// TIA Portal V20 export
FUNCTION_BLOCK "CallEquipment"   // FB32, LAD
TITLE = CallEquipment
AUTHOR : ERsystem_FA2_DH. Kim
// This block contains the logic and futher calls (e.g. sequences, control modules, diagnostics etc.) of the equipment module.
// stored: IsIECCheckEnabled true, MemoryReserve 100, Namespace Unit1.Em4, SetENOAutomatically false
   VAR_INPUT
      ZoneOperationEnable { ExternalWritable := 'False'} : "LWONIK_typeSafetyZoneManualOperation";
   END_VAR
   VAR_IN_OUT
      unitStatus : "LAF_typeUnitStatus";   // Current unit status o be used in this EM
      unitAlarmDB : "LAF_typeAlarms";   // Summarized EM Alarms for the Unit
      emFeedback : "LUC_typeEmFeedback";   // Feedback of the EM to the Unit
   END_VAR
   VAR
      InstSequenceMainPnP : "Unit1.Em4.Sequence_1_MainPnP";   // EM Sequence Instance
      InstSequenceAlignTable : "Unit1.Em4.Sequence_2_AlignTable";
      InstSequenceNgPnP : "Unit1.Em4.Sequence_3_NgPnP";
      InstSequenceGaugeRnR : "Unit1.Em4.Sequence_10_GaugeRnR";
      instMainPnPHomeJob1 : "LAF_SelectJob";
      instMainPnPHomeJob10 : "LAF_SelectJob";
      instMainPnPLoadJob2 : "LAF_SelectJob";
      instMainPnPUnloadJob3 : "LAF_SelectJob";
      instMainPnPAvoidJob4 : "LAF_SelectJob";
      instMainPnPOneLoadJob5 : "LAF_SelectJob";
      instMainPnPOneUnLoadJob6 : "LAF_SelectJob";
      instMainPnPDownWaitJob7 { S7_SetPoint := 'True'} : "LAF_SelectJob";
      instAlignTableHomeJob1 : "LAF_SelectJob";
      instAlignTableLoadJob2 : "LAF_SelectJob";
      instAlignTableVisionJob3 : "LAF_SelectJob";
      instAlignTableUnloadJob4 : "LAF_SelectJob";
      instAlignTableMotionJob22 : "LAF_SelectJob";
      instNgPnPHomeJob1 : "LAF_SelectJob";
      instNgPnPLoadJob2 : "LAF_SelectJob";
      instNgPnPUnloadJob3 : "LAF_SelectJob";
      instGaugeRnRCommonReadyJob1 : "LAF_SelectJob";
      instGaugeRnRCommonGetMasterPieceJob2 : "LAF_SelectJob";
      instGaugeRnRCommonMainPnPMoveAlignTableStackTableJob3 : "LAF_SelectJob";
      instGaugeRnRCommonMainPnp1ToAlignTableJob4 : "LAF_SelectJob";
      instGaugeRnRCommonMainPnPMoveReelCutConvyorAlignTableJob5 : "LAF_SelectJob";
      instGaugeRnRCommonAlignTableVisionAdjustJob6 : "LAF_SelectJob";
      instGaugeRnR1AlignAlignTableToMainPnP1Job10 { S7_SetPoint := 'True'} : "LAF_SelectJob";
      instGaugeRnR1AlignMainPnPMoveReelCutConvyorAlignTableJob11 { S7_SetPoint := 'True'} : "LAF_SelectJob";
      instGaugeRnR1AlignAlignTableMoveWaitJob12 { S7_SetPoint := 'True'} : "LAF_SelectJob";
      instGaugeRnR1AlignUnloadMasterPieceJob13 { S7_SetPoint := 'True'} : "LAF_SelectJob";
      instGaugeRnR1StackMainPnPMoveReelCutConvyorAlignTableJob15 { S7_SetPoint := 'True'} : "LAF_SelectJob";
      instGaugeRnR1StackAlignTableToMainPnP2Job16 { S7_SetPoint := 'True'} : "LAF_SelectJob";
      instGaugeRnR1StackMainPnPMoveAlignTableJob17 { S7_SetPoint := 'True'} : "LAF_SelectJob";
      instGaugeRnR1StackAlignTableMoveWaitJob18 { S7_SetPoint := 'True'} : "LAF_SelectJob";
      instGaugeRnR1StackMainPnP2ToStackTableJob19 { S7_SetPoint := 'True'} : "LAF_SelectJob";
      instGaugeRnR1StackStackTableToMainPnP2Job20 { S7_SetPoint := 'True'} : "LAF_SelectJob";
      instGaugeRnR1StackMainPnPMoveReelCutConvyorAlignTableJob21 { S7_SetPoint := 'True'} : "LAF_SelectJob";
      instGaugeRnR1StackMainPnP2ToAlignTableJob22 { S7_SetPoint := 'True'} : "LAF_SelectJob";
      instGaugeRnR1StackMainPnPMoveAlignTableJob23 { S7_SetPoint := 'True'} : "LAF_SelectJob";
      instGaugeRnR1StackAlignTableToMainPnP1Job24 { S7_SetPoint := 'True'} : "LAF_SelectJob";
      instGaugeRnR1StackMainPnPMoveReelCutConvyorAlignTableJob25 { S7_SetPoint := 'True'} : "LAF_SelectJob";
      instGaugeRnR1StackUnloadMasterPieceJob26 { S7_SetPoint := 'True'} : "LAF_SelectJob";
      instGaugeRnR3AlignMainPnPMoveReelCutConvyorAlignTableJob30 { S7_SetPoint := 'True'} : "LAF_SelectJob";
      instGaugeRnR3AlignNGPnPLoadMasterPieceJob31 { S7_SetPoint := 'True'} : "LAF_SelectJob";
      instGaugeRnR3AlignMainPnP2MoveAlignTableJob32 { S7_SetPoint := 'True'} : "LAF_SelectJob";
      instGaugeRnR3AlignAlignTableMoveWaitJob33 { S7_SetPoint := 'True'} : "LAF_SelectJob";
      instGaugeRnRCommonCheckCompleteJob39 { S7_SetPoint := 'True'} : "LAF_SelectJob";
      instCmPnp1stAnodeDetectSensor { S7_SetPoint := 'True'} : "LBC_DigitalSignalCn";
      instCmPnp2ndAnodeDetectSensor { S7_SetPoint := 'True'} : "LBC_DigitalSignalCn";
      instCmAnodeAlignTableElectrodeDetectSensor { S7_SetPoint := 'True'} : "LBC_DigitalSignalCn";
      instCmAnodeNgBoxFullSensorDetectSensor { S7_SetPoint := 'True'} : "LBC_DigitalSignalCn";
      instCmAnodeNgBoxDetectSensor { S7_SetPoint := 'True'} : "LBC_DigitalSignalCn";
      instCmAnodeMainPnP1AxisX { S7_SetPoint := 'True'} : "LBC_Axis64Pos_TecPlcCn";   // Axis 64Position Function Block
      instCmAnodeMainPnP2AxisX { S7_SetPoint := 'True'} : "LBC_Axis64Pos_TecPlcCn";   // Axis 64Position Function Block
      instCmAnodeMainPnP1AxisY { S7_SetPoint := 'True'} : "LBC_Axis64Pos_TecPlcCn";   // Axis 64Position Function Block
      instCmAnodeMainPnP1AxisZ { S7_SetPoint := 'True'} : "LBC_Axis64Pos_TecPlcCn";   // Axis 64Position Function Block
      instCmAnodeMainPnP2AxisZ { S7_SetPoint := 'True'} : "LBC_Axis64Pos_TecPlcCn";   // Axis 64Position Function Block
      instCmAnodeAlignTableAxisX { S7_SetPoint := 'True'} : "LBC_Axis64Pos_TecPlcCn";   // Axis 64Position Function Block
      instCmAnodeAlignTableAxisY1 { S7_SetPoint := 'True'} : "LBC_Axis64Pos_TecPlcCn";   // Axis 64Position Function Block
      instCmAnodeAlignTableAxisY2 { S7_SetPoint := 'True'} : "LBC_Axis64Pos_TecPlcCn";   // Axis 64Position Function Block
      instInterlockAnodeMainPnP1AxisX { S7_SetPoint := 'True'} : "LER_Axis64Pos_InterlockSummary";
      instInterlockAnodeMainPnP1AxisY { S7_SetPoint := 'True'} : "LER_Axis64Pos_InterlockSummary";
      instInterlockAnodeMainPnP1AxisZ { S7_SetPoint := 'True'} : "LER_Axis64Pos_InterlockSummary";
      instInterlockAnodeMainPnP2AxisX { S7_SetPoint := 'True'} : "LER_Axis64Pos_InterlockSummary";
      instInterlockAnodeMainPnP2AxisZ { S7_SetPoint := 'True'} : "LER_Axis64Pos_InterlockSummary";
      instInterlockAnodeAlignTableAxisX { S7_SetPoint := 'True'} : "LER_Axis64Pos_InterlockSummary";
      instInterlockAnodeAlignTableAxisY1 { S7_SetPoint := 'True'} : "LER_Axis64Pos_InterlockSummary";
      instInterlockAnodeAlignTableAxisY2 { S7_SetPoint := 'True'} : "LER_Axis64Pos_InterlockSummary";
      instAnodeMainPnP1AxisXSoftCam : "LER_SoftCam_Interface";
      instAnodeMainPnP2AxisXSoftCam { S7_SetPoint := 'True'} : "LER_SoftCam_Interface";
      instAnodeMainPnP1AxisYSoftCam { S7_SetPoint := 'True'} : "LER_SoftCam_Interface";
      instAnodeMainPnP1AxisZSoftCam { S7_SetPoint := 'True'} : "LER_SoftCam_Interface";
      instAnodeMainPnP2AxisZSoftCam { S7_SetPoint := 'True'} : "LER_SoftCam_Interface";
      instAnodeAlignTableAxisXSoftCam { S7_SetPoint := 'True'} : "LER_SoftCam_Interface";
      instAnodeAlignTableAxisY1SoftCam { S7_SetPoint := 'True'} : "LER_SoftCam_Interface";
      instAnodeAlignTableAxisY2SoftCam { S7_SetPoint := 'True'} : "LER_SoftCam_Interface";
      instCmAnodeMainPnP1RotaryCwCcw { ExternalAccessible := 'False'; ExternalVisible := 'False'; ExternalWritable := 'False'} : "LBC_TwoWayActuatorCn";
      instCmAnodeMainPnP1stSuctionPlateVacuum { ExternalAccessible := 'False'; ExternalVisible := 'False'; ExternalWritable := 'False'} : "LBC_TwoWayActuatorCn";
      instCmAnodeMainPnP2ndSuctionPlateVacuum { ExternalAccessible := 'False'; ExternalVisible := 'False'; ExternalWritable := 'False'} : "LBC_TwoWayActuatorCn";
      instCmAnodeAlignTableSuctionPlateVacuum { ExternalAccessible := 'False'; ExternalVisible := 'False'; ExternalWritable := 'False'; S7_SetPoint := 'True'} : "LBC_TwoWayActuatorCn";
      instCmAnodeGlassCleaning { ExternalAccessible := 'False'; ExternalVisible := 'False'; ExternalWritable := 'False'; S7_SetPoint := 'True'} : "LBC_TwoWayActuatorCn";
      instCmAnodeNgPnpUpDown { ExternalAccessible := 'False'; ExternalVisible := 'False'; ExternalWritable := 'False'; S7_SetPoint := 'True'} : "LBC_TwoWayActuatorCn";
      instCmAnodeNgPnp1stFwdBwd { ExternalAccessible := 'False'; ExternalVisible := 'False'; ExternalWritable := 'False'; S7_SetPoint := 'True'} : "LBC_TwoWayActuatorCn";
      instCmAnodeNgPnp2ndFwdBwd { ExternalAccessible := 'False'; ExternalVisible := 'False'; ExternalWritable := 'False'; S7_SetPoint := 'True'} : "LBC_TwoWayActuatorCn";
      instCmAnodeMaintenanceMovingFixFwdBwd { ExternalAccessible := 'False'; ExternalVisible := 'False'; ExternalWritable := 'False'; S7_SetPoint := 'True'} : "LBC_TwoWayActuatorCn";
      instCmAnodeNgBoxLiftUpDown { ExternalAccessible := 'False'; ExternalVisible := 'False'; ExternalWritable := 'False'; S7_SetPoint := 'True'} : "LBC_TwoWayActuatorCn";
      instCmAnodeNgBoxLockUpDown { ExternalAccessible := 'False'; ExternalVisible := 'False'; ExternalWritable := 'False'; S7_SetPoint := 'True'} : "LBC_TwoWayActuatorCn";
      instCmAnodeNgPnpVaccum { ExternalAccessible := 'False'; ExternalVisible := 'False'; ExternalWritable := 'False'; S7_SetPoint := 'True'} : "LBC_TwoWayActuatorCn";
      instCmAnodeConveyorCoverFwdBwd { S7_SetPoint := 'True'} : "LBC_TwoWayActuatorCn";
      instCmAnodeConveyorPickUpBlower { S7_SetPoint := 'True'} : "LBC_TwoWayActuatorCn";
      instCmAnodeVisionControllerInterface { ExternalAccessible := 'False'; ExternalVisible := 'False'; ExternalWritable := 'False'; S7_SetPoint := 'True'} : "LER_Vision_XGX2000";
      instAlignVisionConversion : "LER_AlignVisionConversion";
      instManageAlarms { ExternalWritable := 'False'} : "LAF_ManageAlarms";
      instLER_BrakeTestAnodeMainPnP1AxisZ : "LER_BrakeTest";
      instLER_BrakeTestAnodeMainPnP2AxisZ { S7_SetPoint := 'True'} : "LER_BrakeTest";
      instEventsPFE : "Unit1.Em4.EventsPFE";
      statUnitStatus { ExternalWritable := 'False'} : "LAF_typeUnitStatus";   // Unit Status used in this EM
      statSlmStatus { ExternalWritable := 'False'} : Struct
         running : Bool;
         powerOff : Bool;
      END_STRUCT;
      statAllBrakeTest { ExternalWritable := 'False'} : "LER_typeBrakeTestUnitCommands";
      statInterlockTonTime { ExternalAccessible := 'False'; ExternalVisible := 'False'; ExternalWritable := 'False'} : Struct
         mainPnP1AxisX : Array[0..15] of TON_TIME;
         mainPnP1AxisY : Array[0..15] of TON_TIME;
         mainPnP1AxisZ : Array[0..15] of TON_TIME;
         mainPnP2AxisX : Array[0..15] of TON_TIME;
         mainPnP2AxisZ : Array[0..15] of TON_TIME;
         alignTableAxisX : Array[0..15] of TON_TIME;
         alignTableAxisY1 : Array[0..15] of TON_TIME;
         alignTableAxisY2 : Array[0..15] of TON_TIME;
      END_STRUCT;
      statTonTime { ExternalAccessible := 'False'; ExternalVisible := 'False'; ExternalWritable := 'False'} : Array[0..1999] of TON_TIME;
      statTofTime { ExternalAccessible := 'False'; ExternalVisible := 'False'; ExternalWritable := 'False'} : Array[0..99] of TOF_TIME;
      statPulse { ExternalAccessible := 'False'; ExternalVisible := 'False'; ExternalWritable := 'False'} : Struct
         miscellaneous : Array[0..99] of Bool;
         workingDone : Struct
            mainPnP : Array[0..99] of Bool;
            alignTable : Array[0..99] of Bool;
            ngPnP : Array[0..99] of Bool;
         END_STRUCT;
         axisEnable : Array[0..99] of Bool;
         brakeTest : Array[0..99] of Bool;
      END_STRUCT;
      statEnableManualCmds : Bool;
      Scan_on : Bool;
      "*** Interlock Axis ***" { ExternalAccessible := 'False'; ExternalVisible := 'False'; ExternalWritable := 'False'} : Bool;
      "AnodeMainPnP1AxisX Home" { S7_SetPoint := 'True'} : "Homing.LER_Axis";
      "AnodeMainPnP1AxisX Jog_CW" { S7_SetPoint := 'True'} : "Jog.LER_Axis";
      "AnodeMainPnP1AxisX Jog_CCW" { S7_SetPoint := 'True'} : "Jog.LER_Axis";
      "AnodeMainPnP1AxisX Position_" { S7_SetPoint := 'True'} : Array[0..5] of "Position.LER_Axis";
      "AnodeMainPnP2AxisX Home" { S7_SetPoint := 'True'} : "Homing.LER_Axis";
      "AnodeMainPnP2AxisX Jog_CW" { S7_SetPoint := 'True'} : "Jog.LER_Axis";
      "AnodeMainPnP2AxisX Jog_CCW" { S7_SetPoint := 'True'} : "Jog.LER_Axis";
      "AnodeMainPnP2AxisX Position_" { S7_SetPoint := 'True'} : Array[0..5] of "Position.LER_Axis";
      "AnodeMainPnP1AxisY Home" { S7_SetPoint := 'True'} : "Homing.LER_Axis";
      "AnodeMainPnP1AxisY Jog_CW" { S7_SetPoint := 'True'} : "Jog.LER_Axis";
      "AnodeMainPnP1AxisY Jog_CCW" { S7_SetPoint := 'True'} : "Jog.LER_Axis";
      "AnodeMainPnP1AxisY Position_" { S7_SetPoint := 'True'} : Array[0..5] of "Position.LER_Axis";
      "AnodeMainPnP1AxisZ Home" { S7_SetPoint := 'True'} : "Homing.LER_Axis";
      "AnodeMainPnP1AxisZ Jog_CW" { S7_SetPoint := 'True'} : "Jog.LER_Axis";
      "AnodeMainPnP1AxisZ Jog_CCW" { S7_SetPoint := 'True'} : "Jog.LER_Axis";
      "AnodeMainPnP1AxisZ Position_" { S7_SetPoint := 'True'} : Array[0..5] of "Position.LER_Axis";
      "AnodeMainPnP2AxisZ Home" { S7_SetPoint := 'True'} : "Homing.LER_Axis";
      "AnodeMainPnP2AxisZ Jog_CW" { S7_SetPoint := 'True'} : "Jog.LER_Axis";
      "AnodeMainPnP2AxisZ Jog_CCW" { S7_SetPoint := 'True'} : "Jog.LER_Axis";
      "AnodeMainPnP2AxisZ Position_" { S7_SetPoint := 'True'} : Array[0..5] of "Position.LER_Axis";
      "AnodeAlignTableAxisX Home" { S7_SetPoint := 'True'} : "Homing.LER_Axis";
      "AnodeAlignTableAxisX Jog_CW" { S7_SetPoint := 'True'} : "Jog.LER_Axis";
      "AnodeAlignTableAxisX Jog_CCW" { S7_SetPoint := 'True'} : "Jog.LER_Axis";
      "AnodeAlignTableAxisX Position_" { S7_SetPoint := 'True'} : Array[0..5] of "Position.LER_Axis";
      "AnodeAlignTableAxisY1 Home" { S7_SetPoint := 'True'} : "Homing.LER_Axis";
      "AnodeAlignTableAxisY1 Jog_CW" { S7_SetPoint := 'True'} : "Jog.LER_Axis";
      "AnodeAlignTableAxisY1 Jog_CCW" { S7_SetPoint := 'True'} : "Jog.LER_Axis";
      "AnodeAlignTableAxisY1 Position_" { S7_SetPoint := 'True'} : Array[0..5] of "Position.LER_Axis";
      "AnodeAlignTableAxisY2 Home" { S7_SetPoint := 'True'} : "Homing.LER_Axis";
      "AnodeAlignTableAxisY2 Jog_CW" { S7_SetPoint := 'True'} : "Jog.LER_Axis";
      "AnodeAlignTableAxisY2 Jog_CCW" { S7_SetPoint := 'True'} : "Jog.LER_Axis";
      "AnodeAlignTableAxisY2 Position_" { S7_SetPoint := 'True'} : Array[0..5] of "Position.LER_Axis";
      "*** Interlock Actuator ******" { ExternalAccessible := 'False'; ExternalVisible := 'False'; ExternalWritable := 'False'} : Bool;
      "AnodeNgBoxLiftUpDown Home" { S7_SetPoint := 'True'} : "Cylinder.LER_Actuator";
      "AnodeNgBoxLiftUpDown Work" { S7_SetPoint := 'True'} : "Cylinder.LER_Actuator";
      "AnodeNgBoxLockUpDown Home" { S7_SetPoint := 'True'} : "Cylinder.LER_Actuator";
      "AnodeNgBoxLockUpDown Work" { S7_SetPoint := 'True'} : "Cylinder.LER_Actuator";
      "AnodeMaintenanceMovingFixFrontFwdBwd Home" { S7_SetPoint := 'True'} : "Cylinder.LER_Actuator";
      "AnodeMaintenanceMovingFixFrontFwdBwd Work" { S7_SetPoint := 'True'} : "Cylinder.LER_Actuator";
      "AnodeGlassCleaning Home" { S7_SetPoint := 'True'} : "Cylinder.LER_Actuator";
      "AnodeGlassCleaning Work" { S7_SetPoint := 'True'} : "Cylinder.LER_Actuator";
      "AnodeNgPnp1stFwdBwd Home" { S7_SetPoint := 'True'} : "Cylinder.LER_Actuator";
      "AnodeNgPnp1stFwdBwd Work" { S7_SetPoint := 'True'} : "Cylinder.LER_Actuator";
      "AnodeNgPnpUpDown Home" { S7_SetPoint := 'True'} : "Cylinder.LER_Actuator";
      "AnodeNgPnpUpDown Work" { S7_SetPoint := 'True'} : "Cylinder.LER_Actuator";
      "AnodeMainPnP1RotaryCwCcw Home" { S7_SetPoint := 'True'} : "Cylinder.LER_Actuator";
      "AnodeMainPnP1RotaryCwCcw Work" { S7_SetPoint := 'True'} : "Cylinder.LER_Actuator";
      "AnodeNgPnp2ndFwdBwd Home" { S7_SetPoint := 'True'} : "Cylinder.LER_Actuator";
      "AnodeNgPnp2ndFwdBwd Work" { S7_SetPoint := 'True'} : "Cylinder.LER_Actuator";
      Tracking_04 { S7_SetPoint := 'True'} : "Unit1.Em4.PartData";
      AXIS5 : "LER_CM_Name";
      AXIS11 : "LER_CM_Name";
      AXIS14 : "LER_CM_Name";
      Cylinder13 : "LER_CM_Name";
      Cylinder18 : "LER_CM_Name";
      Vaccum10 : "LER_CM_Name";
      instAlignVisionHistory { S7_SetPoint := 'True'} : "LER_visionHistory";
      instAlignMoveCalibration { S7_SetPoint := 'True'} : "LER_AlignMoveCalibration";
      instAlignThetaCalibration { S7_SetPoint := 'True'} : "LER_AlignThetaCalibration";
      instAlignSyncMove { S7_SetPoint := 'True'} : "LER_AlignSyncMove";
      citi_Ptrig : Array[0..20] of Bool;
      citiTon : Array[0..20] of TON_TIME;
      citi : Time;
      citiTest : Array[0..20] of Bool;
   END_VAR
   VAR_TEMP
      tempIndex : Int;
      tempScInProduction : Bool;   // Mode Production and StateComplete
      tempScNoProduction : Bool;   // Mode Manual and StateComplete
      JogActive : Bool;   // Job Current Active
   END_VAR
   VAR CONSTANT
      delayTime : Time := T#3s;
      TRUE : Bool := TRUE;
      FALSE : Bool := FALSE;
      NO_JOB : DInt;   // No job
      MIN_POSITION_NUMBER : SInt;
      INIT_POSITION_NUMBER : SInt := -1;
   END_VAR
   // // statPulse.brakeTest[0] : Unit Mode Production Rising Edge
   // // statPulse.brakeTest[1] : Unit Mode Production Rising Edge Old
   // // statPulse.brakeTest[10] : Anode Main PnP 1 Z Axis Error Pulse
   // // statPulse.brakeTest[11] : Anode Main PnP 2 Z Axis Error Pulse
   VAR_TEMP   // added for the SCL form of the ladder/FBD networks
      _w1 : Bool;
      _w2 : Bool;
      _w3 : Bool;
      _w4 : Bool;
      _w5 : Bool;
      _w6 : Bool;
      _w7 : Bool;
      _w8 : Bool;
      _w9 : Bool;
      _w10 : Bool;
      _w11 : Bool;
      _w12 : Bool;
      _w13 : Bool;
      _w14 : Bool;
      _w15 : Bool;
   END_VAR
BEGIN

REGION Network 1: BLOCK INFO HEADER
   // (company) / (C) Copyright (year)
   // ---------------------------------------------------------------------------------
   // Title:                             (Title of this block)
   // Comment/Function: (that is implemented in the block)
   // Library/Family:           (that the source is dedicated to)
   // Author:                        (department / person in charge / contact)
   // Target System:          (test system with FW version)
   // Engineering:              TIA Portal (SW version)
   // Restrictions:               (OB types, etc.)
   // Requirements:           (hardware, technological package, etc.)
   // ---------------------------------------------------------------------------------
   // Change log table:
   // Version          | Date             | Signature      | Expert in charge  | Changes applied ------------------------|----------------------|-------------------------|--------------------------------|-----------------------
   // 001.000.000 | yyyy-mm-dd | 0x00000000 | (name of expert) | First released version
END_REGION

REGION Network 2: DESCRIPTION
   // This is a template block provided by the Automation Framework. It can be used to create an own project.
   // The Block Info Header is prepared to put in your own data.
   // Description of the block could be added here and the docu created by Code2Docu.
END_REGION

REGION Network 3: ******************** Unit Input ********************
END_REGION

REGION Network 4: Em6 Relations Softcam
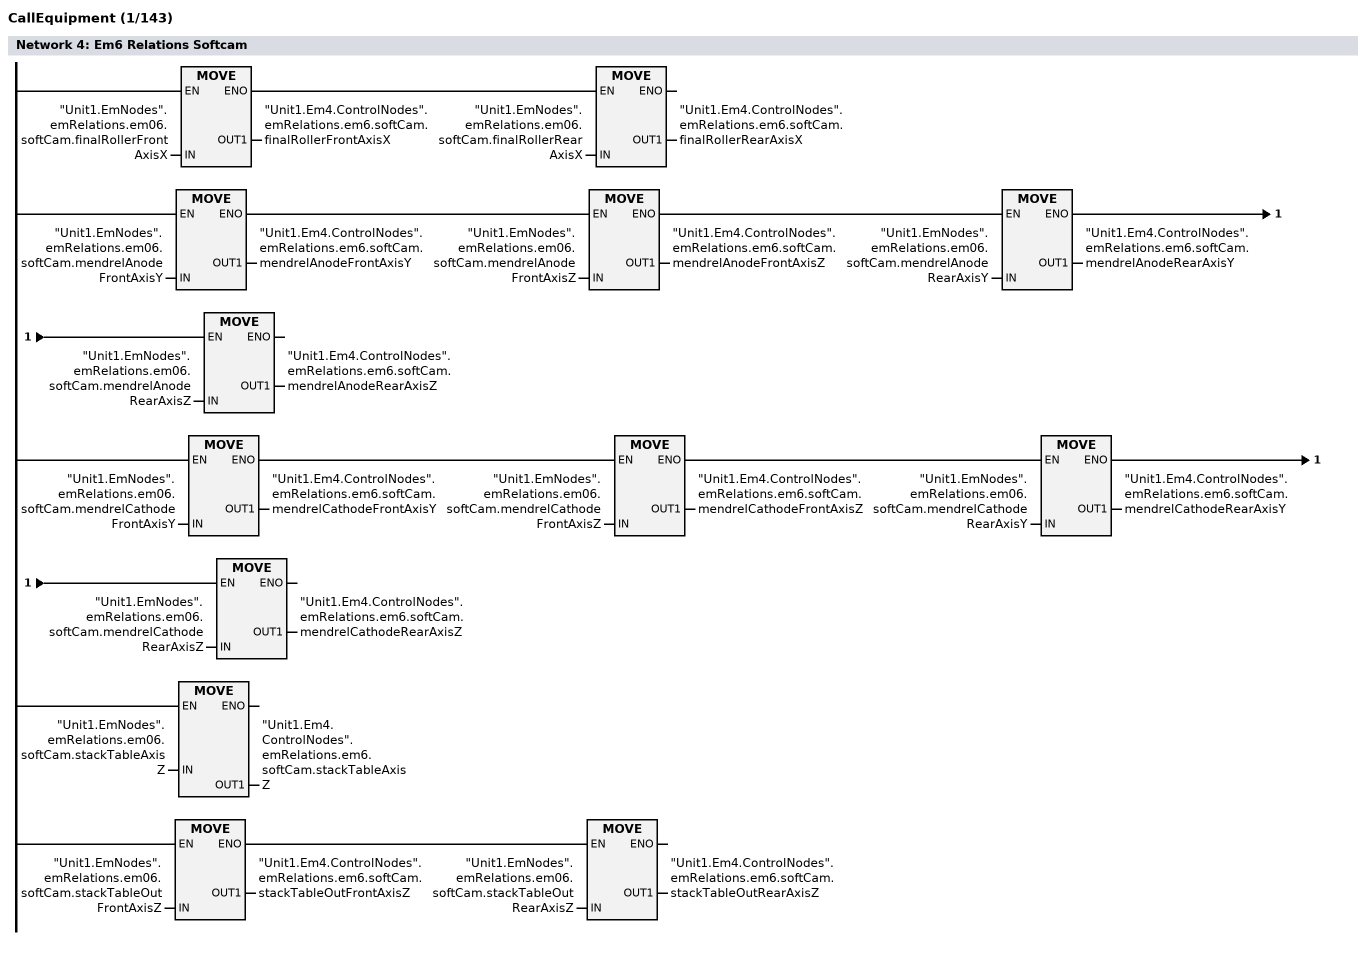
   RUNG wire#powerrail
      Move(in := "Unit1.EmNodes".emRelations.em06.softCam.finalRollerFrontAxisX, out1 => "Unit1.Em4.ControlNodes".emRelations.em6.softCam.finalRollerFrontAxisX)
      Move(in := "Unit1.EmNodes".emRelations.em06.softCam.finalRollerRearAxisX, out1 => "Unit1.Em4.ControlNodes".emRelations.em6.softCam.finalRollerRearAxisX)
   END_RUNG
   RUNG wire#powerrail
      Move(in := "Unit1.EmNodes".emRelations.em06.softCam.mendrelAnodeFrontAxisY, out1 => "Unit1.Em4.ControlNodes".emRelations.em6.softCam.mendrelAnodeFrontAxisY)
      Move(in := "Unit1.EmNodes".emRelations.em06.softCam.mendrelAnodeFrontAxisZ, out1 => "Unit1.Em4.ControlNodes".emRelations.em6.softCam.mendrelAnodeFrontAxisZ)
      Move(in := "Unit1.EmNodes".emRelations.em06.softCam.mendrelAnodeRearAxisY, out1 => "Unit1.Em4.ControlNodes".emRelations.em6.softCam.mendrelAnodeRearAxisY)
      Move(in := "Unit1.EmNodes".emRelations.em06.softCam.mendrelAnodeRearAxisZ, out1 => "Unit1.Em4.ControlNodes".emRelations.em6.softCam.mendrelAnodeRearAxisZ)
   END_RUNG
   RUNG wire#powerrail
      Move(in := "Unit1.EmNodes".emRelations.em06.softCam.mendrelCathodeFrontAxisY, out1 => "Unit1.Em4.ControlNodes".emRelations.em6.softCam.mendrelCathodeFrontAxisY)
      Move(in := "Unit1.EmNodes".emRelations.em06.softCam.mendrelCathodeFrontAxisZ, out1 => "Unit1.Em4.ControlNodes".emRelations.em6.softCam.mendrelCathodeFrontAxisZ)
      Move(in := "Unit1.EmNodes".emRelations.em06.softCam.mendrelCathodeRearAxisY, out1 => "Unit1.Em4.ControlNodes".emRelations.em6.softCam.mendrelCathodeRearAxisY)
      Move(in := "Unit1.EmNodes".emRelations.em06.softCam.mendrelCathodeRearAxisZ, out1 => "Unit1.Em4.ControlNodes".emRelations.em6.softCam.mendrelCathodeRearAxisZ)
   END_RUNG
   RUNG wire#powerrail
      Move(in := "Unit1.EmNodes".emRelations.em06.softCam.stackTableAxisZ, out1 => "Unit1.Em4.ControlNodes".emRelations.em6.softCam.stackTableAxisZ)
   END_RUNG
   RUNG wire#powerrail
      Move(in := "Unit1.EmNodes".emRelations.em06.softCam.stackTableOutFrontAxisZ, out1 => "Unit1.Em4.ControlNodes".emRelations.em6.softCam.stackTableOutFrontAxisZ)
      Move(in := "Unit1.EmNodes".emRelations.em06.softCam.stackTableOutRearAxisZ, out1 => "Unit1.Em4.ControlNodes".emRelations.em6.softCam.stackTableOutRearAxisZ)
   END_RUNG
   // the same network as SCL:
   "Unit1.Em4.ControlNodes".emRelations.em6.softCam.finalRollerFrontAxisX := "Unit1.EmNodes".emRelations.em06.softCam.finalRollerFrontAxisX;
   "Unit1.Em4.ControlNodes".emRelations.em6.softCam.finalRollerRearAxisX := "Unit1.EmNodes".emRelations.em06.softCam.finalRollerRearAxisX;
   "Unit1.Em4.ControlNodes".emRelations.em6.softCam.mendrelAnodeFrontAxisY := "Unit1.EmNodes".emRelations.em06.softCam.mendrelAnodeFrontAxisY;
   "Unit1.Em4.ControlNodes".emRelations.em6.softCam.mendrelAnodeFrontAxisZ := "Unit1.EmNodes".emRelations.em06.softCam.mendrelAnodeFrontAxisZ;
   "Unit1.Em4.ControlNodes".emRelations.em6.softCam.mendrelAnodeRearAxisY := "Unit1.EmNodes".emRelations.em06.softCam.mendrelAnodeRearAxisY;
   "Unit1.Em4.ControlNodes".emRelations.em6.softCam.mendrelAnodeRearAxisZ := "Unit1.EmNodes".emRelations.em06.softCam.mendrelAnodeRearAxisZ;
   "Unit1.Em4.ControlNodes".emRelations.em6.softCam.mendrelCathodeFrontAxisY := "Unit1.EmNodes".emRelations.em06.softCam.mendrelCathodeFrontAxisY;
   "Unit1.Em4.ControlNodes".emRelations.em6.softCam.mendrelCathodeFrontAxisZ := "Unit1.EmNodes".emRelations.em06.softCam.mendrelCathodeFrontAxisZ;
   "Unit1.Em4.ControlNodes".emRelations.em6.softCam.mendrelCathodeRearAxisY := "Unit1.EmNodes".emRelations.em06.softCam.mendrelCathodeRearAxisY;
   "Unit1.Em4.ControlNodes".emRelations.em6.softCam.mendrelCathodeRearAxisZ := "Unit1.EmNodes".emRelations.em06.softCam.mendrelCathodeRearAxisZ;
   "Unit1.Em4.ControlNodes".emRelations.em6.softCam.stackTableAxisZ := "Unit1.EmNodes".emRelations.em06.softCam.stackTableAxisZ;
   "Unit1.Em4.ControlNodes".emRelations.em6.softCam.stackTableOutFrontAxisZ := "Unit1.EmNodes".emRelations.em06.softCam.stackTableOutFrontAxisZ;
   "Unit1.Em4.ControlNodes".emRelations.em6.softCam.stackTableOutRearAxisZ := "Unit1.EmNodes".emRelations.em06.softCam.stackTableOutRearAxisZ;
END_REGION

REGION Network 5: Em7 Relations Softcam
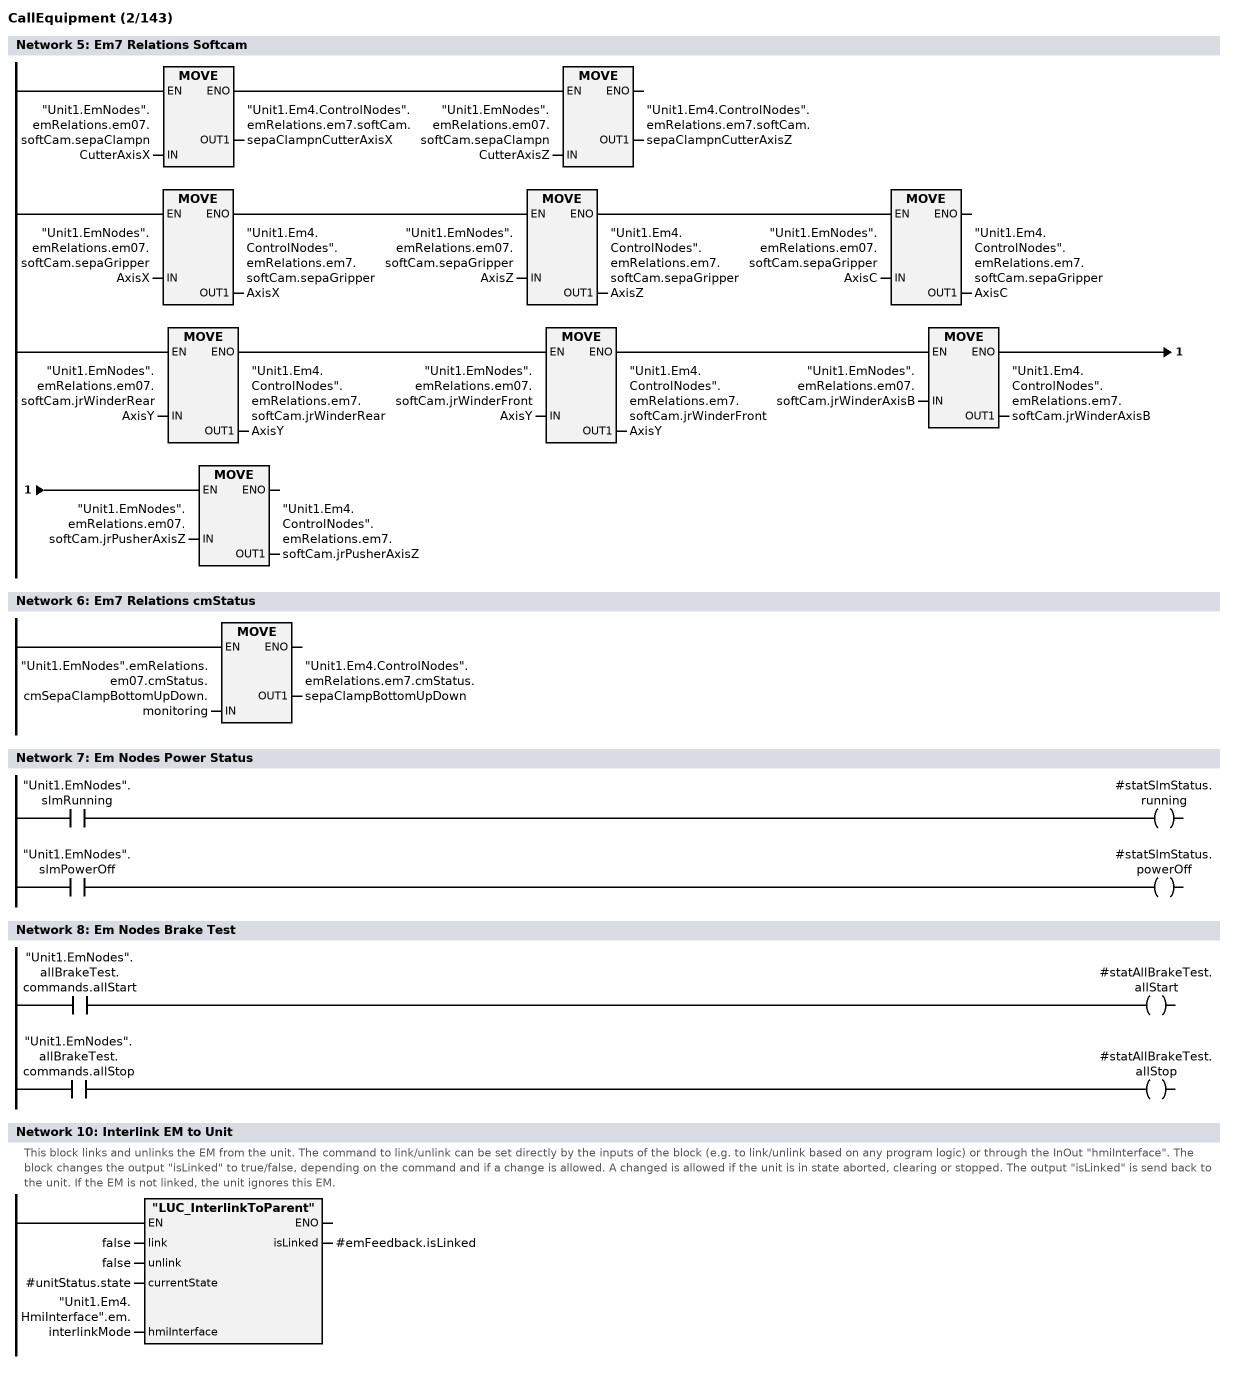
   RUNG wire#powerrail
      Move(in := "Unit1.EmNodes".emRelations.em07.softCam.sepaClampnCutterAxisX, out1 => "Unit1.Em4.ControlNodes".emRelations.em7.softCam.sepaClampnCutterAxisX)
      Move(in := "Unit1.EmNodes".emRelations.em07.softCam.sepaClampnCutterAxisZ, out1 => "Unit1.Em4.ControlNodes".emRelations.em7.softCam.sepaClampnCutterAxisZ)
   END_RUNG
   RUNG wire#powerrail
      Move(in := "Unit1.EmNodes".emRelations.em07.softCam.sepaGripperAxisX, out1 => "Unit1.Em4.ControlNodes".emRelations.em7.softCam.sepaGripperAxisX)
      Move(in := "Unit1.EmNodes".emRelations.em07.softCam.sepaGripperAxisZ, out1 => "Unit1.Em4.ControlNodes".emRelations.em7.softCam.sepaGripperAxisZ)
      Move(in := "Unit1.EmNodes".emRelations.em07.softCam.sepaGripperAxisC, out1 => "Unit1.Em4.ControlNodes".emRelations.em7.softCam.sepaGripperAxisC)
   END_RUNG
   RUNG wire#powerrail
      Move(in := "Unit1.EmNodes".emRelations.em07.softCam.jrWinderRearAxisY, out1 => "Unit1.Em4.ControlNodes".emRelations.em7.softCam.jrWinderRearAxisY)
      Move(in := "Unit1.EmNodes".emRelations.em07.softCam.jrWinderFrontAxisY, out1 => "Unit1.Em4.ControlNodes".emRelations.em7.softCam.jrWinderFrontAxisY)
      Move(in := "Unit1.EmNodes".emRelations.em07.softCam.jrWinderAxisB, out1 => "Unit1.Em4.ControlNodes".emRelations.em7.softCam.jrWinderAxisB)
      Move(in := "Unit1.EmNodes".emRelations.em07.softCam.jrPusherAxisZ, out1 => "Unit1.Em4.ControlNodes".emRelations.em7.softCam.jrPusherAxisZ)
   END_RUNG
   // the same network as SCL:
   "Unit1.Em4.ControlNodes".emRelations.em7.softCam.sepaClampnCutterAxisX := "Unit1.EmNodes".emRelations.em07.softCam.sepaClampnCutterAxisX;
   "Unit1.Em4.ControlNodes".emRelations.em7.softCam.sepaClampnCutterAxisZ := "Unit1.EmNodes".emRelations.em07.softCam.sepaClampnCutterAxisZ;
   "Unit1.Em4.ControlNodes".emRelations.em7.softCam.sepaGripperAxisX := "Unit1.EmNodes".emRelations.em07.softCam.sepaGripperAxisX;
   "Unit1.Em4.ControlNodes".emRelations.em7.softCam.sepaGripperAxisZ := "Unit1.EmNodes".emRelations.em07.softCam.sepaGripperAxisZ;
   "Unit1.Em4.ControlNodes".emRelations.em7.softCam.sepaGripperAxisC := "Unit1.EmNodes".emRelations.em07.softCam.sepaGripperAxisC;
   "Unit1.Em4.ControlNodes".emRelations.em7.softCam.jrWinderRearAxisY := "Unit1.EmNodes".emRelations.em07.softCam.jrWinderRearAxisY;
   "Unit1.Em4.ControlNodes".emRelations.em7.softCam.jrWinderFrontAxisY := "Unit1.EmNodes".emRelations.em07.softCam.jrWinderFrontAxisY;
   "Unit1.Em4.ControlNodes".emRelations.em7.softCam.jrWinderAxisB := "Unit1.EmNodes".emRelations.em07.softCam.jrWinderAxisB;
   "Unit1.Em4.ControlNodes".emRelations.em7.softCam.jrPusherAxisZ := "Unit1.EmNodes".emRelations.em07.softCam.jrPusherAxisZ;
END_REGION

REGION Network 6: Em7 Relations cmStatus
   RUNG wire#powerrail
      Move(in := "Unit1.EmNodes".emRelations.em07.cmStatus.cmSepaClampBottomUpDown.monitoring, out1 => "Unit1.Em4.ControlNodes".emRelations.em7.cmStatus.sepaClampBottomUpDown)
   END_RUNG
   // the same network as SCL:
   "Unit1.Em4.ControlNodes".emRelations.em7.cmStatus.sepaClampBottomUpDown := "Unit1.EmNodes".emRelations.em07.cmStatus.cmSepaClampBottomUpDown.monitoring;
END_REGION

REGION Network 7: Em Nodes Power Status
   RUNG wire#powerrail
      Contact( "Unit1.EmNodes".slmRunning )
      Coil( #statSlmStatus.running )
   END_RUNG
   RUNG wire#powerrail
      Contact( "Unit1.EmNodes".slmPowerOff )
      Coil( #statSlmStatus.powerOff )
   END_RUNG
   // the same network as SCL:
   #statSlmStatus.running := "Unit1.EmNodes".slmRunning;
   #statSlmStatus.powerOff := "Unit1.EmNodes".slmPowerOff;
END_REGION

REGION Network 8: Em Nodes Brake Test
   RUNG wire#powerrail
      Contact( "Unit1.EmNodes".allBrakeTest.commands.allStart )
      Coil( #statAllBrakeTest.allStart )
   END_RUNG
   RUNG wire#powerrail
      Contact( "Unit1.EmNodes".allBrakeTest.commands.allStop )
      Coil( #statAllBrakeTest.allStop )
   END_RUNG
   // the same network as SCL:
   #statAllBrakeTest.allStart := "Unit1.EmNodes".allBrakeTest.commands.allStart;
   #statAllBrakeTest.allStop := "Unit1.EmNodes".allBrakeTest.commands.allStop;
END_REGION

REGION Network 9: *************** Equipment Control **************************
END_REGION

REGION Network 10: Interlink EM to Unit
   // This block links and unlinks the EM from the unit. The command to link/unlink can be set directly by the inputs of the block (e.g. to link/unlink based on any program logic) or through the InOut "hmiInterface". The block changes the output "isLinked" to true/false, depending on the command and if a change is allowed. A changed is allowed if the unit is in state aborted, clearing or stopped. The output "isLinked" is send back to the unit. If the EM is not linked, the unit ignores this EM.
   RUNG wire#powerrail
      "LUC_InterlinkToParent"(link := false, unlink := false, currentState := #unitStatus.state, hmiInterface := "Unit1.Em4.HmiInterface".em.interlinkMode, isLinked => #emFeedback.isLinked)
   END_RUNG
   // the same network as SCL:
   "LUC_InterlinkToParent"(link := false,
                           unlink := false,
                           currentState := #unitStatus.state,
                           hmiInterface := "Unit1.Em4.HmiInterface".em.interlinkMode,
                           isLinked => #emFeedback.isLinked);
END_REGION

REGION Network 11: Control EM
   // When linked, unitStatus is fully applied to unitStatusUsed.
   // When not linked, only acknowledge and safetyReleased from the unitStatus are applied. A direct EM control by hmiInterface or localInterface is possible.
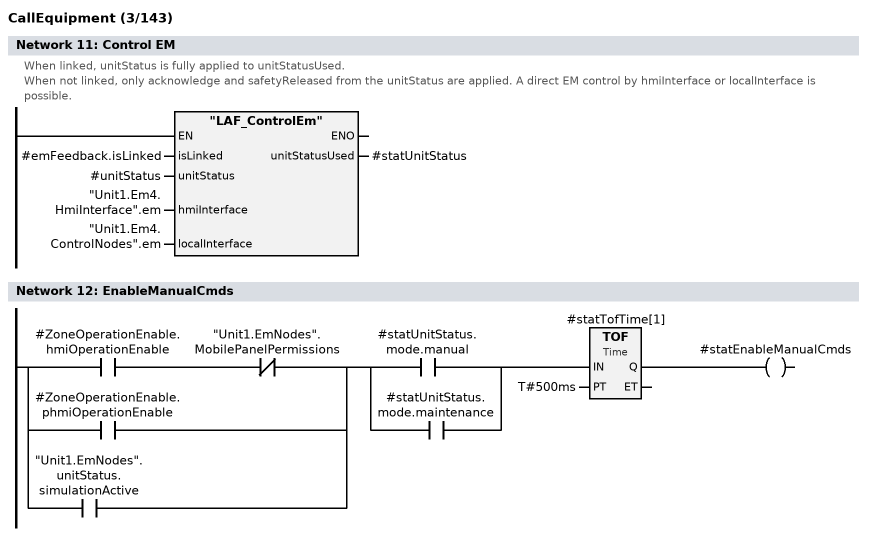
   RUNG wire#powerrail
      "LAF_ControlEm"(isLinked := #emFeedback.isLinked, unitStatus := #unitStatus, hmiInterface := "Unit1.Em4.HmiInterface".em, localInterface := "Unit1.Em4.ControlNodes".em, unitStatusUsed => #statUnitStatus)
   END_RUNG
   // the same network as SCL:
   "LAF_ControlEm"(isLinked := #emFeedback.isLinked,
                   unitStatus := #unitStatus,
                   hmiInterface := "Unit1.Em4.HmiInterface".em,
                   localInterface := "Unit1.Em4.ControlNodes".em,
                   unitStatusUsed => #statUnitStatus);
END_REGION

REGION Network 12: EnableManualCmds
   RUNG wire#powerrail
      Contact( #ZoneOperationEnable.hmiOperationEnable )
      I_Contact( "Unit1.EmNodes".MobilePanelPermissions )
      wire#w1
      Contact( #statUnitStatus.mode.manual )
      wire#w2
      { S7_Templates := "time_type := Time" } #statTofTime[1].TOF(pt := T#500ms, et =>)
      Coil( #statEnableManualCmds )
   END_RUNG
   RUNG wire#powerrail
      Contact( #ZoneOperationEnable.phmiOperationEnable )
   END_RUNG wire#w1
   RUNG wire#powerrail
      Contact( "Unit1.EmNodes".unitStatus.simulationActive )
   END_RUNG wire#w1
   RUNG wire#w1
      Contact( #statUnitStatus.mode.maintenance )
   END_RUNG wire#w2
   // the same network as SCL:
   #statTofTime[1].TOF(IN := ((#ZoneOperationEnable.hmiOperationEnable AND NOT "Unit1.EmNodes".MobilePanelPermissions) OR #ZoneOperationEnable.phmiOperationEnable OR "Unit1.EmNodes".unitStatus.simulationActive) AND (#statUnitStatus.mode.manual OR #statUnitStatus.mode.maintenance),
                       PT := T#500ms);
   #statEnableManualCmds := #statTofTime[1].Q;
END_REGION

REGION Network 13: DryRun Config Setting
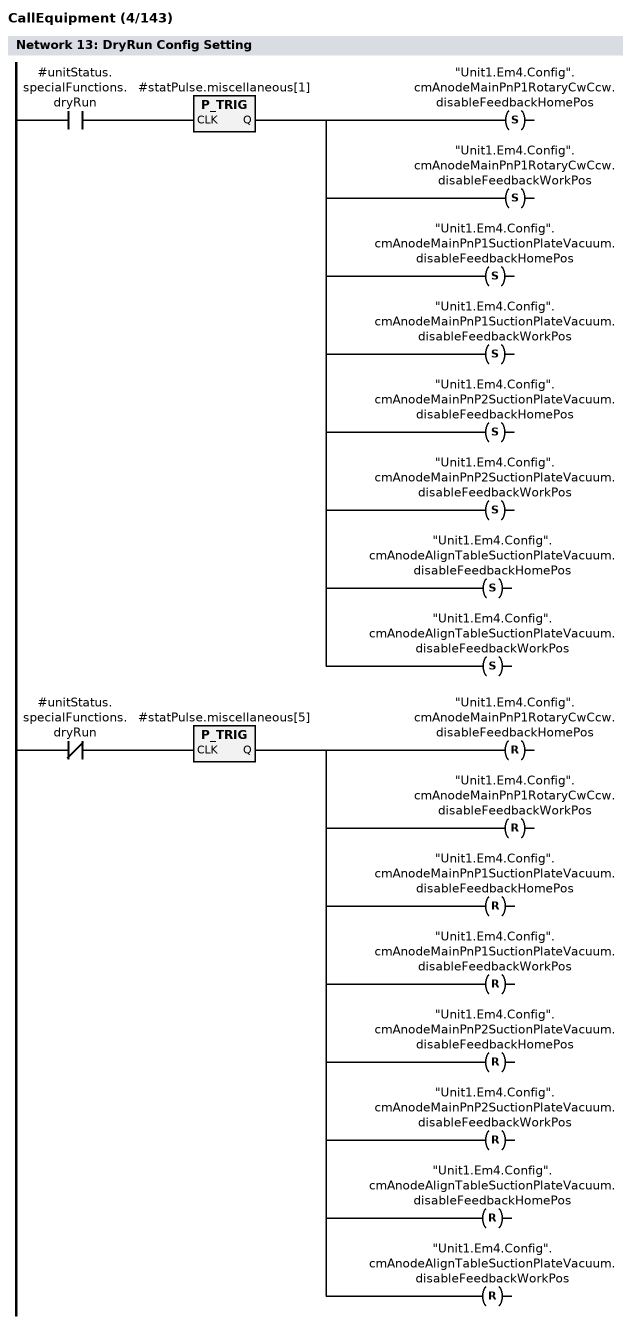
   RUNG wire#powerrail
      Contact( #unitStatus.specialFunctions.dryRun )
      P_Trig( #statPulse.miscellaneous[1] )
      wire#w1
      S_Coil( "Unit1.Em4.Config".cmAnodeMainPnP1RotaryCwCcw.disableFeedbackHomePos )
   END_RUNG
   RUNG wire#w1
      S_Coil( "Unit1.Em4.Config".cmAnodeMainPnP1RotaryCwCcw.disableFeedbackWorkPos )
   END_RUNG
   RUNG wire#w1
      S_Coil( "Unit1.Em4.Config".cmAnodeMainPnP1SuctionPlateVacuum.disableFeedbackHomePos )
   END_RUNG
   RUNG wire#w1
      S_Coil( "Unit1.Em4.Config".cmAnodeMainPnP1SuctionPlateVacuum.disableFeedbackWorkPos )
   END_RUNG
   RUNG wire#w1
      S_Coil( "Unit1.Em4.Config".cmAnodeMainPnP2SuctionPlateVacuum.disableFeedbackHomePos )
   END_RUNG
   RUNG wire#w1
      S_Coil( "Unit1.Em4.Config".cmAnodeMainPnP2SuctionPlateVacuum.disableFeedbackWorkPos )
   END_RUNG
   RUNG wire#w1
      S_Coil( "Unit1.Em4.Config".cmAnodeAlignTableSuctionPlateVacuum.disableFeedbackHomePos )
   END_RUNG
   RUNG wire#w1
      S_Coil( "Unit1.Em4.Config".cmAnodeAlignTableSuctionPlateVacuum.disableFeedbackWorkPos )
   END_RUNG
   RUNG wire#powerrail
      I_Contact( #unitStatus.specialFunctions.dryRun )
      P_Trig( #statPulse.miscellaneous[5] )
      wire#w2
      R_Coil( "Unit1.Em4.Config".cmAnodeMainPnP1RotaryCwCcw.disableFeedbackHomePos )
   END_RUNG
   RUNG wire#w2
      R_Coil( "Unit1.Em4.Config".cmAnodeMainPnP1RotaryCwCcw.disableFeedbackWorkPos )
   END_RUNG
   RUNG wire#w2
      R_Coil( "Unit1.Em4.Config".cmAnodeMainPnP1SuctionPlateVacuum.disableFeedbackHomePos )
   END_RUNG
   RUNG wire#w2
      R_Coil( "Unit1.Em4.Config".cmAnodeMainPnP1SuctionPlateVacuum.disableFeedbackWorkPos )
   END_RUNG
   RUNG wire#w2
      R_Coil( "Unit1.Em4.Config".cmAnodeMainPnP2SuctionPlateVacuum.disableFeedbackHomePos )
   END_RUNG
   RUNG wire#w2
      R_Coil( "Unit1.Em4.Config".cmAnodeMainPnP2SuctionPlateVacuum.disableFeedbackWorkPos )
   END_RUNG
   RUNG wire#w2
      R_Coil( "Unit1.Em4.Config".cmAnodeAlignTableSuctionPlateVacuum.disableFeedbackHomePos )
   END_RUNG
   RUNG wire#w2
      R_Coil( "Unit1.Em4.Config".cmAnodeAlignTableSuctionPlateVacuum.disableFeedbackWorkPos )
   END_RUNG
   // the same network as SCL:
   #_w1 := #unitStatus.specialFunctions.dryRun AND NOT #statPulse.miscellaneous[1];   // rising edge
   #statPulse.miscellaneous[1] := #unitStatus.specialFunctions.dryRun;
   IF #_w1 THEN
       "Unit1.Em4.Config".cmAnodeMainPnP1RotaryCwCcw.disableFeedbackHomePos := TRUE;
       "Unit1.Em4.Config".cmAnodeMainPnP1RotaryCwCcw.disableFeedbackWorkPos := TRUE;
       "Unit1.Em4.Config".cmAnodeMainPnP1SuctionPlateVacuum.disableFeedbackHomePos := TRUE;
       "Unit1.Em4.Config".cmAnodeMainPnP1SuctionPlateVacuum.disableFeedbackWorkPos := TRUE;
       "Unit1.Em4.Config".cmAnodeMainPnP2SuctionPlateVacuum.disableFeedbackHomePos := TRUE;
       "Unit1.Em4.Config".cmAnodeMainPnP2SuctionPlateVacuum.disableFeedbackWorkPos := TRUE;
       "Unit1.Em4.Config".cmAnodeAlignTableSuctionPlateVacuum.disableFeedbackHomePos := TRUE;
       "Unit1.Em4.Config".cmAnodeAlignTableSuctionPlateVacuum.disableFeedbackWorkPos := TRUE;
   END_IF;
   #_w2 := NOT #unitStatus.specialFunctions.dryRun AND NOT #statPulse.miscellaneous[5];   // rising edge
   #statPulse.miscellaneous[5] := NOT #unitStatus.specialFunctions.dryRun;
   IF #_w2 THEN
       "Unit1.Em4.Config".cmAnodeMainPnP1RotaryCwCcw.disableFeedbackHomePos := FALSE;
       "Unit1.Em4.Config".cmAnodeMainPnP1RotaryCwCcw.disableFeedbackWorkPos := FALSE;
       "Unit1.Em4.Config".cmAnodeMainPnP1SuctionPlateVacuum.disableFeedbackHomePos := FALSE;
       "Unit1.Em4.Config".cmAnodeMainPnP1SuctionPlateVacuum.disableFeedbackWorkPos := FALSE;
       "Unit1.Em4.Config".cmAnodeMainPnP2SuctionPlateVacuum.disableFeedbackHomePos := FALSE;
       "Unit1.Em4.Config".cmAnodeMainPnP2SuctionPlateVacuum.disableFeedbackWorkPos := FALSE;
       "Unit1.Em4.Config".cmAnodeAlignTableSuctionPlateVacuum.disableFeedbackHomePos := FALSE;
       "Unit1.Em4.Config".cmAnodeAlignTableSuctionPlateVacuum.disableFeedbackWorkPos := FALSE;
   END_IF;
END_REGION

REGION Network 14: *************** Control Modules (Sensors) ********************
   // Call control modules that are sensors before the em logic (jobs and sequence), so that the latest value is used in the logic.
END_REGION

REGION Network 15: Call Pnp1stAnodeDetectSensor (LBC_DigitalSignal)
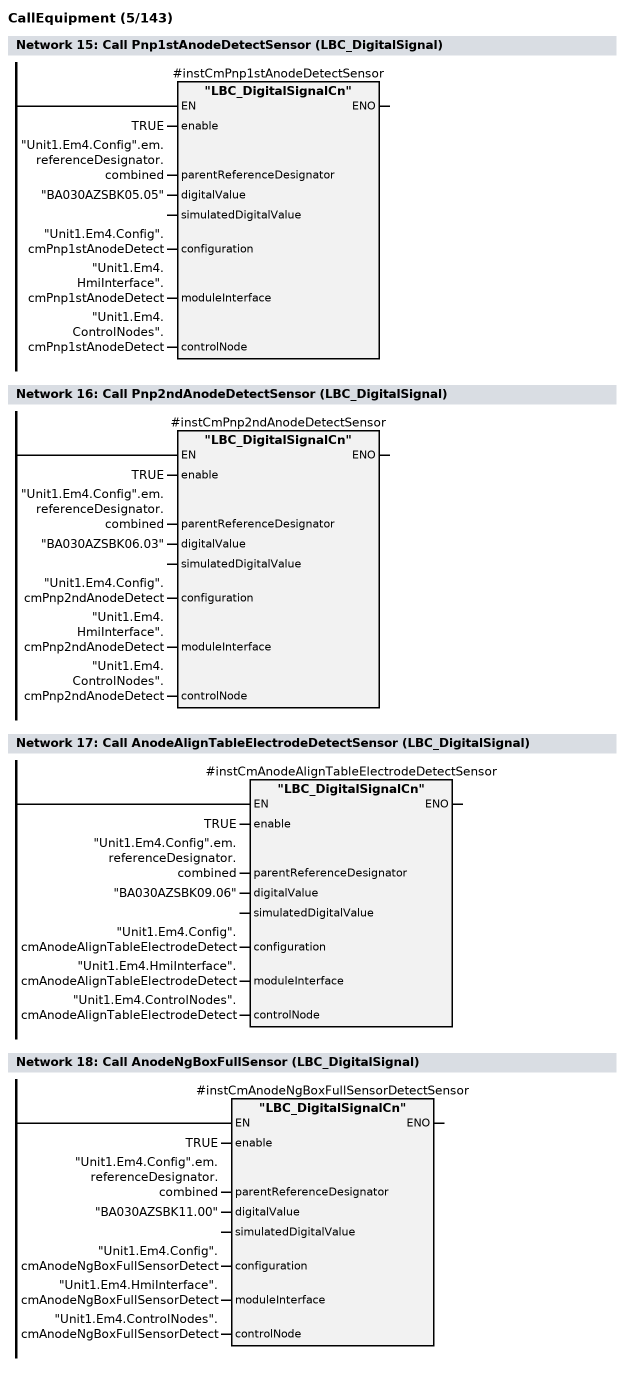
   RUNG wire#powerrail
      #instCmPnp1stAnodeDetectSensor(enable := TRUE, parentReferenceDesignator := "Unit1.Em4.Config".em.referenceDesignator.combined, digitalValue := "BA030AZSBK05.05", simulatedDigitalValue :=, configuration := "Unit1.Em4.Config".cmPnp1stAnodeDetect, moduleInterface := "Unit1.Em4.HmiInterface".cmPnp1stAnodeDetect, controlNode := "Unit1.Em4.ControlNodes".cmPnp1stAnodeDetect)
   END_RUNG
   // the same network as SCL:
   #instCmPnp1stAnodeDetectSensor(enable := TRUE,   // "LBC_DigitalSignalCn"
                           parentReferenceDesignator := "Unit1.Em4.Config".em.referenceDesignator.combined,
                           digitalValue := "BA030AZSBK05.05",
                           configuration := "Unit1.Em4.Config".cmPnp1stAnodeDetect,
                           moduleInterface := "Unit1.Em4.HmiInterface".cmPnp1stAnodeDetect,
                           controlNode := "Unit1.Em4.ControlNodes".cmPnp1stAnodeDetect);
END_REGION

REGION Network 16: Call Pnp2ndAnodeDetectSensor (LBC_DigitalSignal)
   RUNG wire#powerrail
      #instCmPnp2ndAnodeDetectSensor(enable := TRUE, parentReferenceDesignator := "Unit1.Em4.Config".em.referenceDesignator.combined, digitalValue := "BA030AZSBK06.03", simulatedDigitalValue :=, configuration := "Unit1.Em4.Config".cmPnp2ndAnodeDetect, moduleInterface := "Unit1.Em4.HmiInterface".cmPnp2ndAnodeDetect, controlNode := "Unit1.Em4.ControlNodes".cmPnp2ndAnodeDetect)
   END_RUNG
   // the same network as SCL:
   #instCmPnp2ndAnodeDetectSensor(enable := TRUE,   // "LBC_DigitalSignalCn"
                           parentReferenceDesignator := "Unit1.Em4.Config".em.referenceDesignator.combined,
                           digitalValue := "BA030AZSBK06.03",
                           configuration := "Unit1.Em4.Config".cmPnp2ndAnodeDetect,
                           moduleInterface := "Unit1.Em4.HmiInterface".cmPnp2ndAnodeDetect,
                           controlNode := "Unit1.Em4.ControlNodes".cmPnp2ndAnodeDetect);
END_REGION

REGION Network 17: Call AnodeAlignTableElectrodeDetectSensor (LBC_DigitalSignal)
   RUNG wire#powerrail
      #instCmAnodeAlignTableElectrodeDetectSensor(enable := TRUE, parentReferenceDesignator := "Unit1.Em4.Config".em.referenceDesignator.combined, digitalValue := "BA030AZSBK09.06", simulatedDigitalValue :=, configuration := "Unit1.Em4.Config".cmAnodeAlignTableElectrodeDetect, moduleInterface := "Unit1.Em4.HmiInterface".cmAnodeAlignTableElectrodeDetect, controlNode := "Unit1.Em4.ControlNodes".cmAnodeAlignTableElectrodeDetect)
   END_RUNG
   // the same network as SCL:
   #instCmAnodeAlignTableElectrodeDetectSensor(enable := TRUE,   // "LBC_DigitalSignalCn"
                           parentReferenceDesignator := "Unit1.Em4.Config".em.referenceDesignator.combined,
                           digitalValue := "BA030AZSBK09.06",
                           configuration := "Unit1.Em4.Config".cmAnodeAlignTableElectrodeDetect,
                           moduleInterface := "Unit1.Em4.HmiInterface".cmAnodeAlignTableElectrodeDetect,
                           controlNode := "Unit1.Em4.ControlNodes".cmAnodeAlignTableElectrodeDetect);
END_REGION

REGION Network 18: Call AnodeNgBoxFullSensor (LBC_DigitalSignal)
   RUNG wire#powerrail
      #instCmAnodeNgBoxFullSensorDetectSensor(enable := TRUE, parentReferenceDesignator := "Unit1.Em4.Config".em.referenceDesignator.combined, digitalValue := "BA030AZSBK11.00", simulatedDigitalValue :=, configuration := "Unit1.Em4.Config".cmAnodeNgBoxFullSensorDetect, moduleInterface := "Unit1.Em4.HmiInterface".cmAnodeNgBoxFullSensorDetect, controlNode := "Unit1.Em4.ControlNodes".cmAnodeNgBoxFullSensorDetect)
   END_RUNG
   // the same network as SCL:
   #instCmAnodeNgBoxFullSensorDetectSensor(enable := TRUE,   // "LBC_DigitalSignalCn"
                           parentReferenceDesignator := "Unit1.Em4.Config".em.referenceDesignator.combined,
                           digitalValue := "BA030AZSBK11.00",
                           configuration := "Unit1.Em4.Config".cmAnodeNgBoxFullSensorDetect,
                           moduleInterface := "Unit1.Em4.HmiInterface".cmAnodeNgBoxFullSensorDetect,
                           controlNode := "Unit1.Em4.ControlNodes".cmAnodeNgBoxFullSensorDetect);
END_REGION

REGION Network 19: Call AnodeNgBoxDetectSensor (LBC_DigitalSignal)
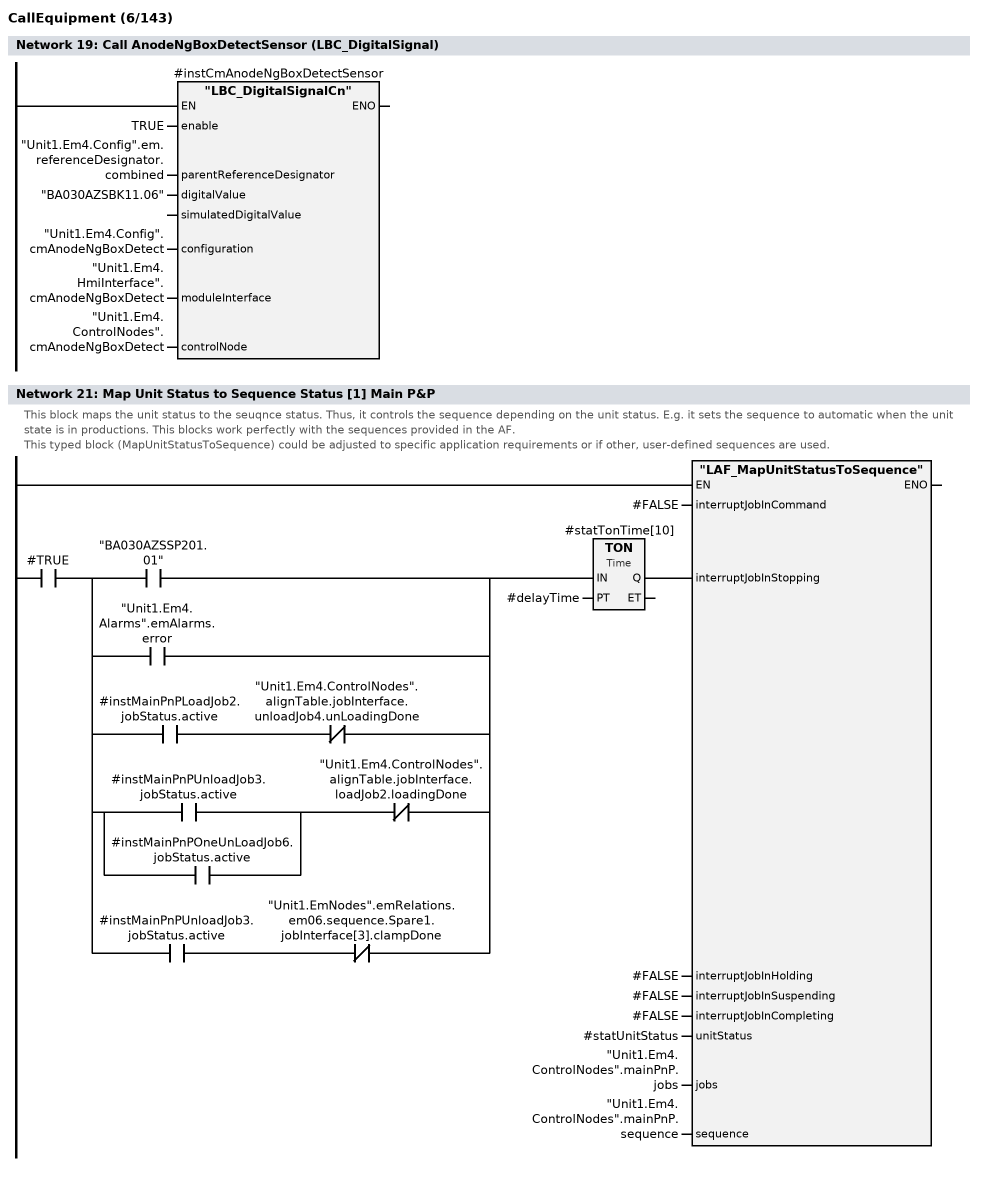
   RUNG wire#powerrail
      #instCmAnodeNgBoxDetectSensor(enable := TRUE, parentReferenceDesignator := "Unit1.Em4.Config".em.referenceDesignator.combined, digitalValue := "BA030AZSBK11.06", simulatedDigitalValue :=, configuration := "Unit1.Em4.Config".cmAnodeNgBoxDetect, moduleInterface := "Unit1.Em4.HmiInterface".cmAnodeNgBoxDetect, controlNode := "Unit1.Em4.ControlNodes".cmAnodeNgBoxDetect)
   END_RUNG
   // the same network as SCL:
   #instCmAnodeNgBoxDetectSensor(enable := TRUE,   // "LBC_DigitalSignalCn"
                           parentReferenceDesignator := "Unit1.Em4.Config".em.referenceDesignator.combined,
                           digitalValue := "BA030AZSBK11.06",
                           configuration := "Unit1.Em4.Config".cmAnodeNgBoxDetect,
                           moduleInterface := "Unit1.Em4.HmiInterface".cmAnodeNgBoxDetect,
                           controlNode := "Unit1.Em4.ControlNodes".cmAnodeNgBoxDetect);
END_REGION

REGION Network 20: *************** Equipment Logic ***************************
END_REGION

REGION Network 21: Map Unit Status to Sequence Status [1] Main P&P
   // This block maps the unit status to the seuqnce status. Thus, it controls the sequence depending on the unit status. E.g. it sets the sequence to automatic when the unit state is in productions. This blocks work perfectly with the sequences provided in the AF. 
   // This typed block (MapUnitStatusToSequence) could be adjusted to specific application requirements or if other, user-defined sequences are used.
   RUNG wire#powerrail
      "LAF_MapUnitStatusToSequence"(interruptJobInStopping := wire#w4, interruptJobInCommand := #FALSE, interruptJobInHolding := #FALSE, interruptJobInSuspending := #FALSE, interruptJobInCompleting := #FALSE, unitStatus := #statUnitStatus, jobs := "Unit1.Em4.ControlNodes".mainPnP.jobs, sequence := "Unit1.Em4.ControlNodes".mainPnP.sequence)
   END_RUNG
   RUNG wire#powerrail
      Contact( #TRUE )
      wire#w1
      Contact( "BA030AZSSP201.01" )
      wire#w2
      { S7_Templates := "time_type := Time" } #statTonTime[10].TON(pt := #delayTime, et =>)
   END_RUNG wire#w4
   RUNG wire#w1
      Contact( "Unit1.Em4.Alarms".emAlarms.error )
   END_RUNG wire#w2
   RUNG wire#w1
      Contact( #instMainPnPLoadJob2.jobStatus.active )
      I_Contact( "Unit1.Em4.ControlNodes".alignTable.jobInterface.unloadJob4.unLoadingDone )
   END_RUNG wire#w2
   RUNG wire#w1
      Contact( #instMainPnPUnloadJob3.jobStatus.active )
      wire#w3
      I_Contact( "Unit1.Em4.ControlNodes".alignTable.jobInterface.loadJob2.loadingDone )
   END_RUNG wire#w2
   RUNG wire#w1
      Contact( #instMainPnPOneUnLoadJob6.jobStatus.active )
   END_RUNG wire#w3
   RUNG wire#w1
      Contact( #instMainPnPUnloadJob3.jobStatus.active )
      I_Contact( "Unit1.EmNodes".emRelations.em06.sequence.Spare1.jobInterface[3].clampDone )
   END_RUNG wire#w2
   // the same network as SCL:
   #statTonTime[10].TON(IN := #TRUE AND ("BA030AZSSP201.01" OR "Unit1.Em4.Alarms".emAlarms.error OR (#instMainPnPLoadJob2.jobStatus.active AND NOT "Unit1.Em4.ControlNodes".alignTable.jobInterface.unloadJob4.unLoadingDone) OR ((#instMainPnPUnloadJob3.jobStatus.active OR #instMainPnPOneUnLoadJob6.jobStatus.active) AND NOT "Unit1.Em4.ControlNodes".alignTable.jobInterface.loadJob2.loadingDone) OR (#instMainPnPUnloadJob3.jobStatus.active AND NOT "Unit1.EmNodes".emRelations.em06.sequence.Spare1.jobInterface[3].clampDone)),
                        PT := #delayTime);
   "LAF_MapUnitStatusToSequence"(interruptJobInCommand := #FALSE,
                           interruptJobInStopping := #statTonTime[10].Q,
                           interruptJobInHolding := #FALSE,
                           interruptJobInSuspending := #FALSE,
                           interruptJobInCompleting := #FALSE,
                           unitStatus := #statUnitStatus,
                           jobs := "Unit1.Em4.ControlNodes".mainPnP.jobs,
                           sequence := "Unit1.Em4.ControlNodes".mainPnP.sequence);
END_REGION

REGION Network 22: Map Unit Status to Sequence Status [2] Align Table
   // This block maps the unit status to the seuqnce status. Thus, it controls the sequence depending on the unit status. E.g. it sets the sequence to automatic when the unit state is in productions. This blocks work perfectly with the sequences provided in the AF. 
   // This typed block (MapUnitStatusToSequence) could be adjusted to specific application requirements or if other, user-defined sequences are used.
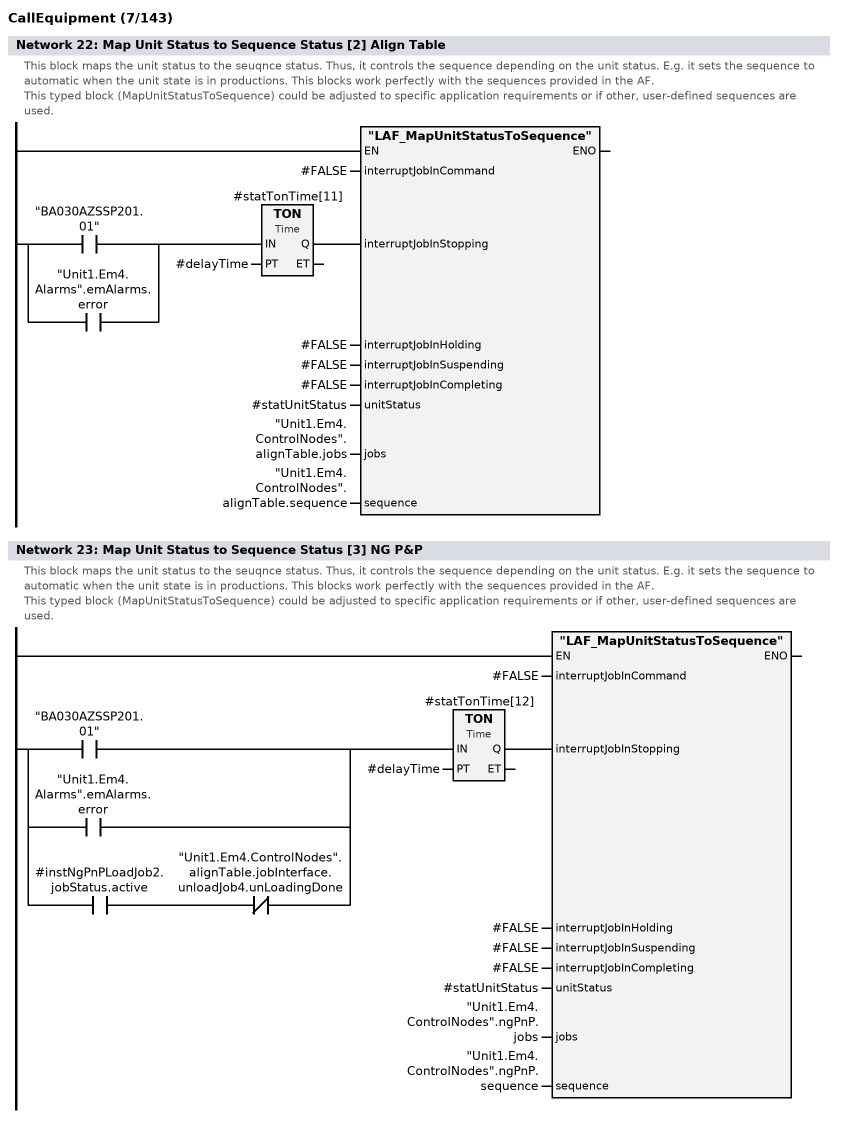
   RUNG wire#powerrail
      "LAF_MapUnitStatusToSequence"(interruptJobInStopping := wire#w2, interruptJobInCommand := #FALSE, interruptJobInHolding := #FALSE, interruptJobInSuspending := #FALSE, interruptJobInCompleting := #FALSE, unitStatus := #statUnitStatus, jobs := "Unit1.Em4.ControlNodes".alignTable.jobs, sequence := "Unit1.Em4.ControlNodes".alignTable.sequence)
   END_RUNG
   RUNG wire#powerrail
      Contact( "BA030AZSSP201.01" )
      wire#w1
      { S7_Templates := "time_type := Time" } #statTonTime[11].TON(pt := #delayTime, et =>)
   END_RUNG wire#w2
   RUNG wire#powerrail
      Contact( "Unit1.Em4.Alarms".emAlarms.error )
   END_RUNG wire#w1
   // the same network as SCL:
   #statTonTime[11].TON(IN := "BA030AZSSP201.01" OR "Unit1.Em4.Alarms".emAlarms.error, PT := #delayTime);
   "LAF_MapUnitStatusToSequence"(interruptJobInCommand := #FALSE,
                           interruptJobInStopping := #statTonTime[11].Q,
                           interruptJobInHolding := #FALSE,
                           interruptJobInSuspending := #FALSE,
                           interruptJobInCompleting := #FALSE,
                           unitStatus := #statUnitStatus,
                           jobs := "Unit1.Em4.ControlNodes".alignTable.jobs,
                           sequence := "Unit1.Em4.ControlNodes".alignTable.sequence);
END_REGION

REGION Network 23: Map Unit Status to Sequence Status [3] NG P&P
   // This block maps the unit status to the seuqnce status. Thus, it controls the sequence depending on the unit status. E.g. it sets the sequence to automatic when the unit state is in productions. This blocks work perfectly with the sequences provided in the AF. 
   // This typed block (MapUnitStatusToSequence) could be adjusted to specific application requirements or if other, user-defined sequences are used.
   RUNG wire#powerrail
      "LAF_MapUnitStatusToSequence"(interruptJobInStopping := wire#w2, interruptJobInCommand := #FALSE, interruptJobInHolding := #FALSE, interruptJobInSuspending := #FALSE, interruptJobInCompleting := #FALSE, unitStatus := #statUnitStatus, jobs := "Unit1.Em4.ControlNodes".ngPnP.jobs, sequence := "Unit1.Em4.ControlNodes".ngPnP.sequence)
   END_RUNG
   RUNG wire#powerrail
      Contact( "BA030AZSSP201.01" )
      wire#w1
      { S7_Templates := "time_type := Time" } #statTonTime[12].TON(pt := #delayTime, et =>)
   END_RUNG wire#w2
   RUNG wire#powerrail
      Contact( "Unit1.Em4.Alarms".emAlarms.error )
   END_RUNG wire#w1
   RUNG wire#powerrail
      Contact( #instNgPnPLoadJob2.jobStatus.active )
      I_Contact( "Unit1.Em4.ControlNodes".alignTable.jobInterface.unloadJob4.unLoadingDone )
   END_RUNG wire#w1
   // the same network as SCL:
   #statTonTime[12].TON(IN := "BA030AZSSP201.01" OR "Unit1.Em4.Alarms".emAlarms.error OR (#instNgPnPLoadJob2.jobStatus.active AND NOT "Unit1.Em4.ControlNodes".alignTable.jobInterface.unloadJob4.unLoadingDone),
                        PT := #delayTime);
   "LAF_MapUnitStatusToSequence"(interruptJobInCommand := #FALSE,
                           interruptJobInStopping := #statTonTime[12].Q,
                           interruptJobInHolding := #FALSE,
                           interruptJobInSuspending := #FALSE,
                           interruptJobInCompleting := #FALSE,
                           unitStatus := #statUnitStatus,
                           jobs := "Unit1.Em4.ControlNodes".ngPnP.jobs,
                           sequence := "Unit1.Em4.ControlNodes".ngPnP.sequence);
END_REGION

REGION Network 24: Map Unit Status to Sequence Status [4] Gague R&R
   // This block maps the unit status to the seuqnce status. Thus, it controls the sequence depending on the unit status. E.g. it sets the sequence to automatic when the unit state is in productions. This blocks work perfectly with the sequences provided in the AF. 
   // This typed block (MapUnitStatusToSequence) could be adjusted to specific application requirements or if other, user-defined sequences are used.
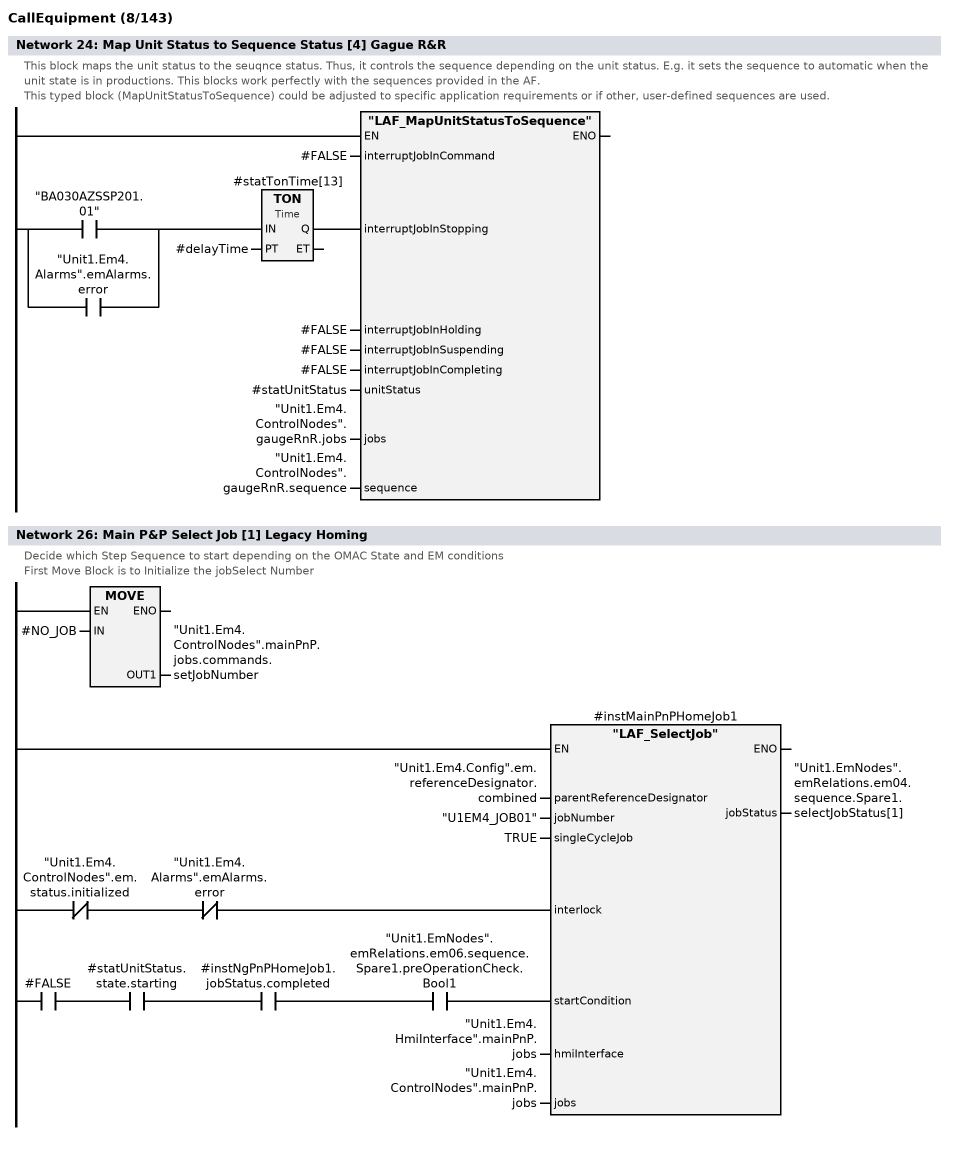
   RUNG wire#powerrail
      "LAF_MapUnitStatusToSequence"(interruptJobInStopping := wire#w2, interruptJobInCommand := #FALSE, interruptJobInHolding := #FALSE, interruptJobInSuspending := #FALSE, interruptJobInCompleting := #FALSE, unitStatus := #statUnitStatus, jobs := "Unit1.Em4.ControlNodes".gaugeRnR.jobs, sequence := "Unit1.Em4.ControlNodes".gaugeRnR.sequence)
   END_RUNG
   RUNG wire#powerrail
      Contact( "BA030AZSSP201.01" )
      wire#w1
      { S7_Templates := "time_type := Time" } #statTonTime[13].TON(pt := #delayTime, et =>)
   END_RUNG wire#w2
   RUNG wire#powerrail
      Contact( "Unit1.Em4.Alarms".emAlarms.error )
   END_RUNG wire#w1
   // the same network as SCL:
   #statTonTime[13].TON(IN := "BA030AZSSP201.01" OR "Unit1.Em4.Alarms".emAlarms.error, PT := #delayTime);
   "LAF_MapUnitStatusToSequence"(interruptJobInCommand := #FALSE,
                           interruptJobInStopping := #statTonTime[13].Q,
                           interruptJobInHolding := #FALSE,
                           interruptJobInSuspending := #FALSE,
                           interruptJobInCompleting := #FALSE,
                           unitStatus := #statUnitStatus,
                           jobs := "Unit1.Em4.ControlNodes".gaugeRnR.jobs,
                           sequence := "Unit1.Em4.ControlNodes".gaugeRnR.sequence);
END_REGION

REGION Network 26: Main P&P Select Job [1] Legacy Homing
   // Decide which Step Sequence to start depending on the OMAC State and EM conditions
   // First Move Block is to Initialize the jobSelect Number
   RUNG wire#powerrail
      Move(in := #NO_JOB, out1 => "Unit1.Em4.ControlNodes".mainPnP.jobs.commands.setJobNumber)
   END_RUNG
   RUNG wire#powerrail
      #instMainPnPHomeJob1(interlock := wire#w1, startCondition := wire#w2, parentReferenceDesignator := "Unit1.Em4.Config".em.referenceDesignator.combined, jobNumber := "U1EM4_JOB01", singleCycleJob := TRUE, hmiInterface := "Unit1.Em4.HmiInterface".mainPnP.jobs, jobs := "Unit1.Em4.ControlNodes".mainPnP.jobs, jobStatus => "Unit1.EmNodes".emRelations.em04.sequence.Spare1.selectJobStatus[1])
   END_RUNG
   RUNG wire#powerrail
      I_Contact( "Unit1.Em4.ControlNodes".em.status.initialized )
      I_Contact( "Unit1.Em4.Alarms".emAlarms.error )
   END_RUNG wire#w1
   RUNG wire#powerrail
      Contact( #FALSE )
      Contact( #statUnitStatus.state.starting )
      Contact( #instNgPnPHomeJob1.jobStatus.completed )
      Contact( "Unit1.EmNodes".emRelations.em06.sequence.Spare1.preOperationCheck.Bool1 )
   END_RUNG wire#w2
   // the same network as SCL:
   "Unit1.Em4.ControlNodes".mainPnP.jobs.commands.setJobNumber := #NO_JOB;
   #instMainPnPHomeJob1(parentReferenceDesignator := "Unit1.Em4.Config".em.referenceDesignator.combined,   // "LAF_SelectJob"
                        jobNumber := "U1EM4_JOB01",
                        singleCycleJob := TRUE,
                        interlock := NOT "Unit1.Em4.ControlNodes".em.status.initialized AND NOT "Unit1.Em4.Alarms".emAlarms.error,
                        startCondition := #FALSE AND #statUnitStatus.state.starting AND #instNgPnPHomeJob1.jobStatus.completed AND "Unit1.EmNodes".emRelations.em06.sequence.Spare1.preOperationCheck.Bool1,
                        hmiInterface := "Unit1.Em4.HmiInterface".mainPnP.jobs,
                        jobs := "Unit1.Em4.ControlNodes".mainPnP.jobs,
                        jobStatus => "Unit1.EmNodes".emRelations.em04.sequence.Spare1.selectJobStatus[1]);
END_REGION

REGION Network 27: Main P&P Select Job [10] Homing
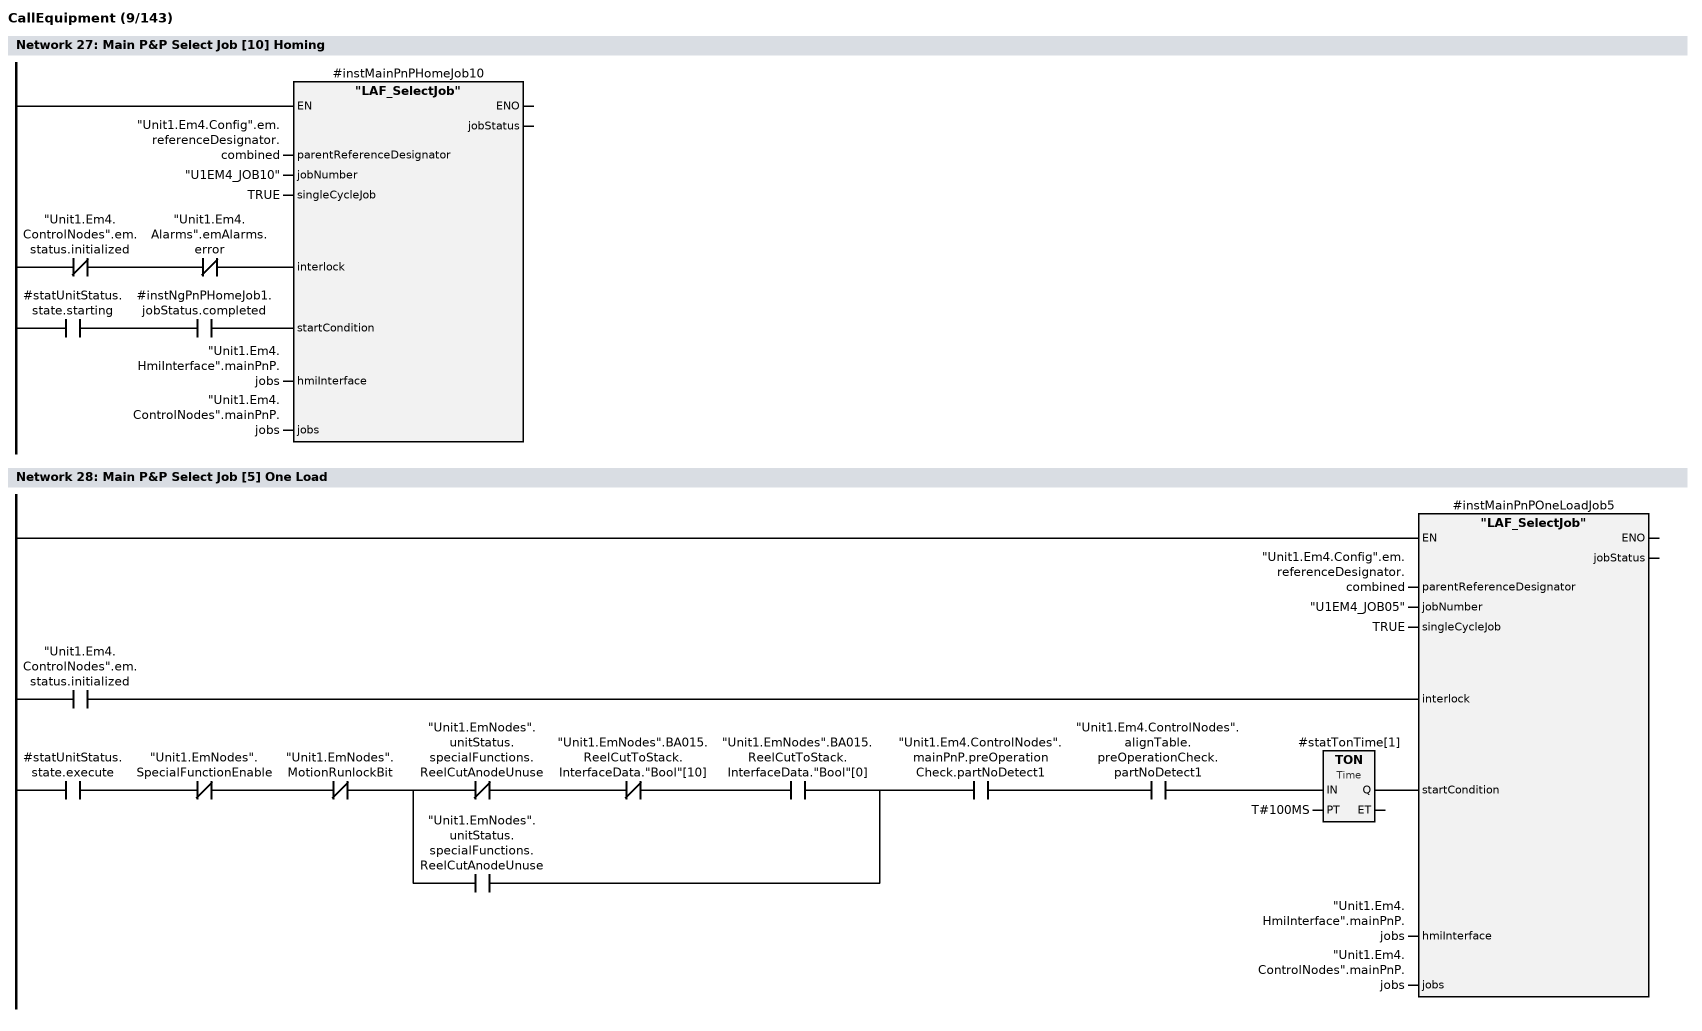
   RUNG wire#powerrail
      #instMainPnPHomeJob10(interlock := wire#w1, startCondition := wire#w2, parentReferenceDesignator := "Unit1.Em4.Config".em.referenceDesignator.combined, jobNumber := "U1EM4_JOB10", singleCycleJob := TRUE, hmiInterface := "Unit1.Em4.HmiInterface".mainPnP.jobs, jobs := "Unit1.Em4.ControlNodes".mainPnP.jobs, jobStatus =>)
   END_RUNG
   RUNG wire#powerrail
      I_Contact( "Unit1.Em4.ControlNodes".em.status.initialized )
      I_Contact( "Unit1.Em4.Alarms".emAlarms.error )
   END_RUNG wire#w1
   RUNG wire#powerrail
      Contact( #statUnitStatus.state.starting )
      Contact( #instNgPnPHomeJob1.jobStatus.completed )
   END_RUNG wire#w2
   // the same network as SCL:
   #instMainPnPHomeJob10(parentReferenceDesignator := "Unit1.Em4.Config".em.referenceDesignator.combined,   // "LAF_SelectJob"
                         jobNumber := "U1EM4_JOB10",
                         singleCycleJob := TRUE,
                         interlock := NOT "Unit1.Em4.ControlNodes".em.status.initialized AND NOT "Unit1.Em4.Alarms".emAlarms.error,
                         startCondition := #statUnitStatus.state.starting AND #instNgPnPHomeJob1.jobStatus.completed,
                         hmiInterface := "Unit1.Em4.HmiInterface".mainPnP.jobs,
                         jobs := "Unit1.Em4.ControlNodes".mainPnP.jobs);
END_REGION

REGION Network 28: Main P&P Select Job [5] One Load
   RUNG wire#powerrail
      #instMainPnPOneLoadJob5(interlock := wire#w1, startCondition := wire#w4, parentReferenceDesignator := "Unit1.Em4.Config".em.referenceDesignator.combined, jobNumber := "U1EM4_JOB05", singleCycleJob := TRUE, hmiInterface := "Unit1.Em4.HmiInterface".mainPnP.jobs, jobs := "Unit1.Em4.ControlNodes".mainPnP.jobs, jobStatus =>)
   END_RUNG
   RUNG wire#powerrail
      Contact( "Unit1.Em4.ControlNodes".em.status.initialized )
   END_RUNG wire#w1
   RUNG wire#powerrail
      Contact( #statUnitStatus.state.execute )
      I_Contact( "Unit1.EmNodes".SpecialFunctionEnable )
      I_Contact( "Unit1.EmNodes".MotionRunlockBit )
      wire#w2
      I_Contact( "Unit1.EmNodes".unitStatus.specialFunctions.ReelCutAnodeUnuse )
      I_Contact( "Unit1.EmNodes".BA015.ReelCutToStack.InterfaceData."Bool"[10] )
      Contact( "Unit1.EmNodes".BA015.ReelCutToStack.InterfaceData."Bool"[0] )
      wire#w3
      Contact( "Unit1.Em4.ControlNodes".mainPnP.preOperationCheck.partNoDetect1 )
      Contact( "Unit1.Em4.ControlNodes".alignTable.preOperationCheck.partNoDetect1 )
      { S7_Templates := "time_type := Time" } #statTonTime[1].TON(pt := T#100MS, et =>)
   END_RUNG wire#w4
   RUNG wire#w2
      Contact( "Unit1.EmNodes".unitStatus.specialFunctions.ReelCutAnodeUnuse )
   END_RUNG wire#w3
   // the same network as SCL:
   #statTonTime[1].TON(IN := #statUnitStatus.state.execute AND NOT "Unit1.EmNodes".SpecialFunctionEnable AND NOT "Unit1.EmNodes".MotionRunlockBit AND ((NOT "Unit1.EmNodes".unitStatus.specialFunctions.ReelCutAnodeUnuse AND NOT "Unit1.EmNodes".BA015.ReelCutToStack.InterfaceData."Bool"[10] AND "Unit1.EmNodes".BA015.ReelCutToStack.InterfaceData."Bool"[0]) OR "Unit1.EmNodes".unitStatus.specialFunctions.ReelCutAnodeUnuse) AND "Unit1.Em4.ControlNodes".mainPnP.preOperationCheck.partNoDetect1 AND "Unit1.Em4.ControlNodes".alignTable.preOperationCheck.partNoDetect1,
                       PT := T#100MS);
   #instMainPnPOneLoadJob5(parentReferenceDesignator := "Unit1.Em4.Config".em.referenceDesignator.combined,   // "LAF_SelectJob"
                           jobNumber := "U1EM4_JOB05",
                           singleCycleJob := TRUE,
                           interlock := "Unit1.Em4.ControlNodes".em.status.initialized,
                           startCondition := #statTonTime[1].Q,
                           hmiInterface := "Unit1.Em4.HmiInterface".mainPnP.jobs,
                           jobs := "Unit1.Em4.ControlNodes".mainPnP.jobs);
END_REGION

REGION Network 29: Main P&P Select Job [6] One UnLoad
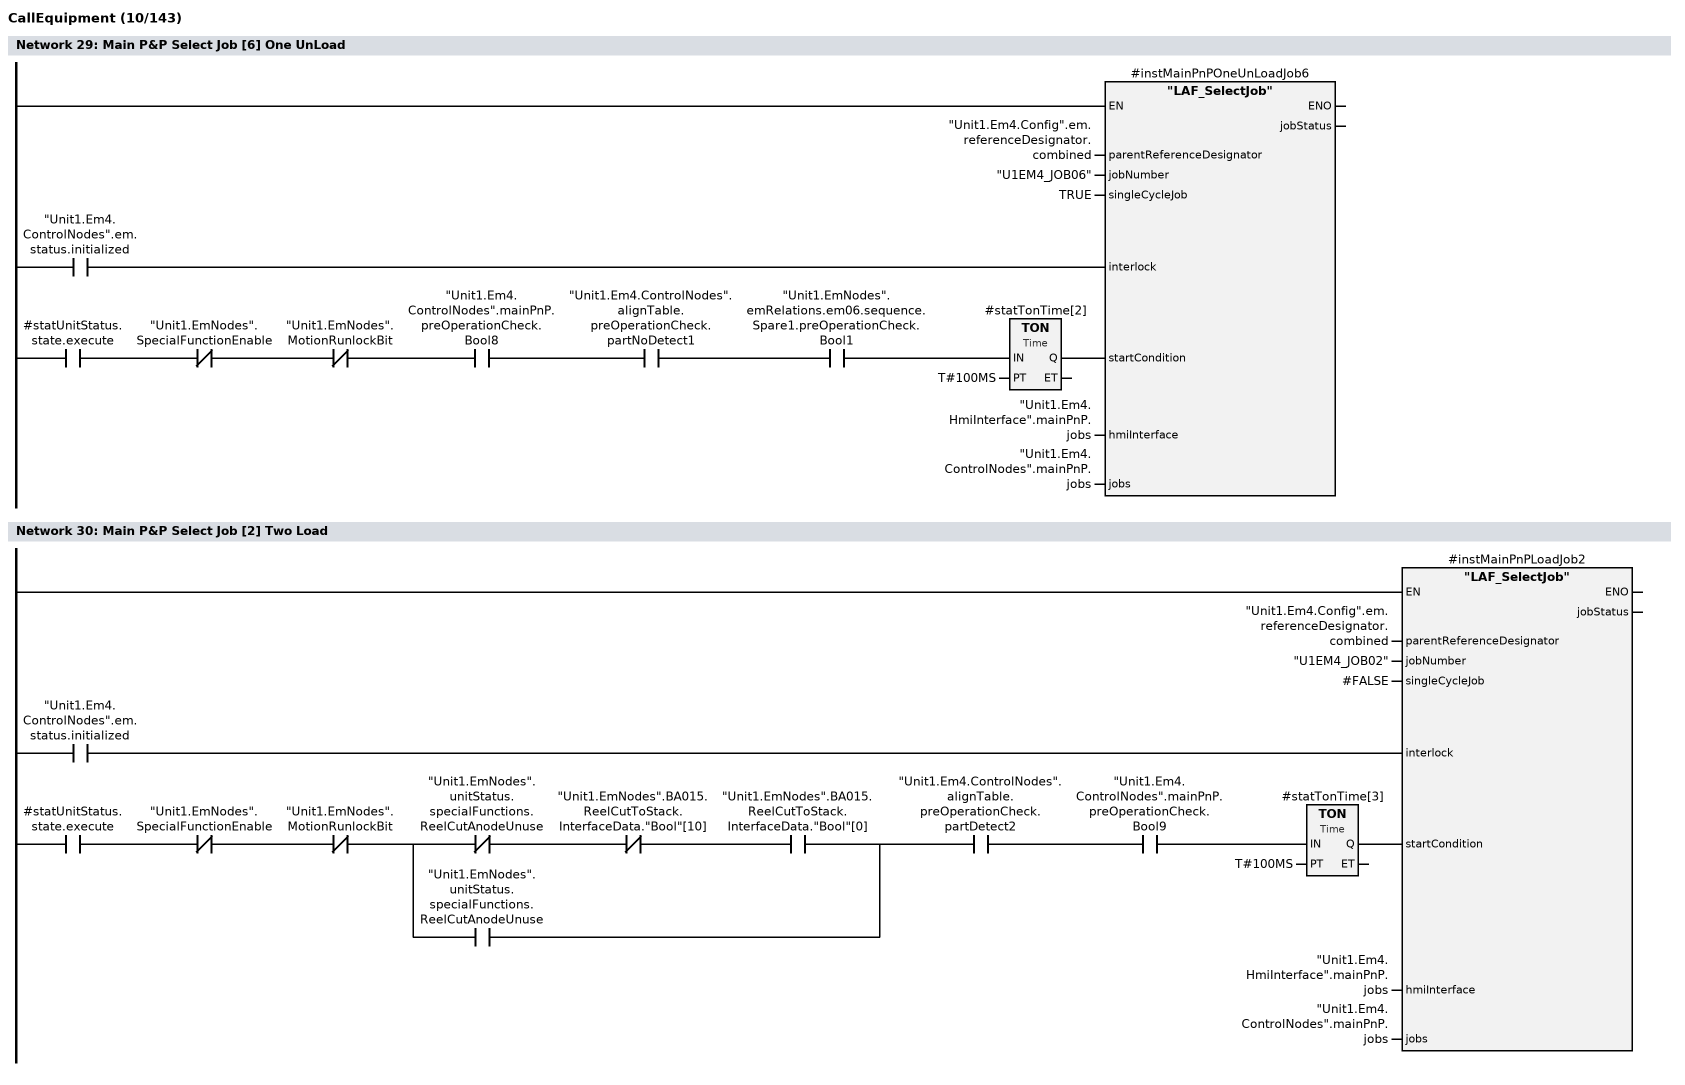
   RUNG wire#powerrail
      #instMainPnPOneUnLoadJob6(interlock := wire#w1, startCondition := wire#w2, parentReferenceDesignator := "Unit1.Em4.Config".em.referenceDesignator.combined, jobNumber := "U1EM4_JOB06", singleCycleJob := TRUE, hmiInterface := "Unit1.Em4.HmiInterface".mainPnP.jobs, jobs := "Unit1.Em4.ControlNodes".mainPnP.jobs, jobStatus =>)
   END_RUNG
   RUNG wire#powerrail
      Contact( "Unit1.Em4.ControlNodes".em.status.initialized )
   END_RUNG wire#w1
   RUNG wire#powerrail
      Contact( #statUnitStatus.state.execute )
      I_Contact( "Unit1.EmNodes".SpecialFunctionEnable )
      I_Contact( "Unit1.EmNodes".MotionRunlockBit )
      Contact( "Unit1.Em4.ControlNodes".mainPnP.preOperationCheck.Bool8 )
      Contact( "Unit1.Em4.ControlNodes".alignTable.preOperationCheck.partNoDetect1 )
      Contact( "Unit1.EmNodes".emRelations.em06.sequence.Spare1.preOperationCheck.Bool1 )
      { S7_Templates := "time_type := Time" } #statTonTime[2].TON(pt := T#100MS, et =>)
   END_RUNG wire#w2
   // the same network as SCL:
   #statTonTime[2].TON(IN := #statUnitStatus.state.execute AND NOT "Unit1.EmNodes".SpecialFunctionEnable AND NOT "Unit1.EmNodes".MotionRunlockBit AND "Unit1.Em4.ControlNodes".mainPnP.preOperationCheck.Bool8 AND "Unit1.Em4.ControlNodes".alignTable.preOperationCheck.partNoDetect1 AND "Unit1.EmNodes".emRelations.em06.sequence.Spare1.preOperationCheck.Bool1,
                       PT := T#100MS);
   #instMainPnPOneUnLoadJob6(parentReferenceDesignator := "Unit1.Em4.Config".em.referenceDesignator.combined,   // "LAF_SelectJob"
                           jobNumber := "U1EM4_JOB06",
                           singleCycleJob := TRUE,
                           interlock := "Unit1.Em4.ControlNodes".em.status.initialized,
                           startCondition := #statTonTime[2].Q,
                           hmiInterface := "Unit1.Em4.HmiInterface".mainPnP.jobs,
                           jobs := "Unit1.Em4.ControlNodes".mainPnP.jobs);
END_REGION

REGION Network 30: Main P&P Select Job [2] Two Load
   RUNG wire#powerrail
      #instMainPnPLoadJob2(interlock := wire#w1, startCondition := wire#w4, parentReferenceDesignator := "Unit1.Em4.Config".em.referenceDesignator.combined, jobNumber := "U1EM4_JOB02", singleCycleJob := #FALSE, hmiInterface := "Unit1.Em4.HmiInterface".mainPnP.jobs, jobs := "Unit1.Em4.ControlNodes".mainPnP.jobs, jobStatus =>)
   END_RUNG
   RUNG wire#powerrail
      Contact( "Unit1.Em4.ControlNodes".em.status.initialized )
   END_RUNG wire#w1
   RUNG wire#powerrail
      Contact( #statUnitStatus.state.execute )
      I_Contact( "Unit1.EmNodes".SpecialFunctionEnable )
      I_Contact( "Unit1.EmNodes".MotionRunlockBit )
      wire#w2
      I_Contact( "Unit1.EmNodes".unitStatus.specialFunctions.ReelCutAnodeUnuse )
      I_Contact( "Unit1.EmNodes".BA015.ReelCutToStack.InterfaceData."Bool"[10] )
      Contact( "Unit1.EmNodes".BA015.ReelCutToStack.InterfaceData."Bool"[0] )
      wire#w3
      Contact( "Unit1.Em4.ControlNodes".alignTable.preOperationCheck.partDetect2 )
      Contact( "Unit1.Em4.ControlNodes".mainPnP.preOperationCheck.Bool9 )
      { S7_Templates := "time_type := Time" } #statTonTime[3].TON(pt := T#100MS, et =>)
   END_RUNG wire#w4
   RUNG wire#w2
      Contact( "Unit1.EmNodes".unitStatus.specialFunctions.ReelCutAnodeUnuse )
   END_RUNG wire#w3
   // the same network as SCL:
   #statTonTime[3].TON(IN := #statUnitStatus.state.execute AND NOT "Unit1.EmNodes".SpecialFunctionEnable AND NOT "Unit1.EmNodes".MotionRunlockBit AND ((NOT "Unit1.EmNodes".unitStatus.specialFunctions.ReelCutAnodeUnuse AND NOT "Unit1.EmNodes".BA015.ReelCutToStack.InterfaceData."Bool"[10] AND "Unit1.EmNodes".BA015.ReelCutToStack.InterfaceData."Bool"[0]) OR "Unit1.EmNodes".unitStatus.specialFunctions.ReelCutAnodeUnuse) AND "Unit1.Em4.ControlNodes".alignTable.preOperationCheck.partDetect2 AND "Unit1.Em4.ControlNodes".mainPnP.preOperationCheck.Bool9,
                       PT := T#100MS);
   #instMainPnPLoadJob2(parentReferenceDesignator := "Unit1.Em4.Config".em.referenceDesignator.combined,   // "LAF_SelectJob"
                        jobNumber := "U1EM4_JOB02",
                        singleCycleJob := #FALSE,
                        interlock := "Unit1.Em4.ControlNodes".em.status.initialized,
                        startCondition := #statTonTime[3].Q,
                        hmiInterface := "Unit1.Em4.HmiInterface".mainPnP.jobs,
                        jobs := "Unit1.Em4.ControlNodes".mainPnP.jobs);
END_REGION

REGION Network 31: Main P&P Select Job [3] Two UnLoad
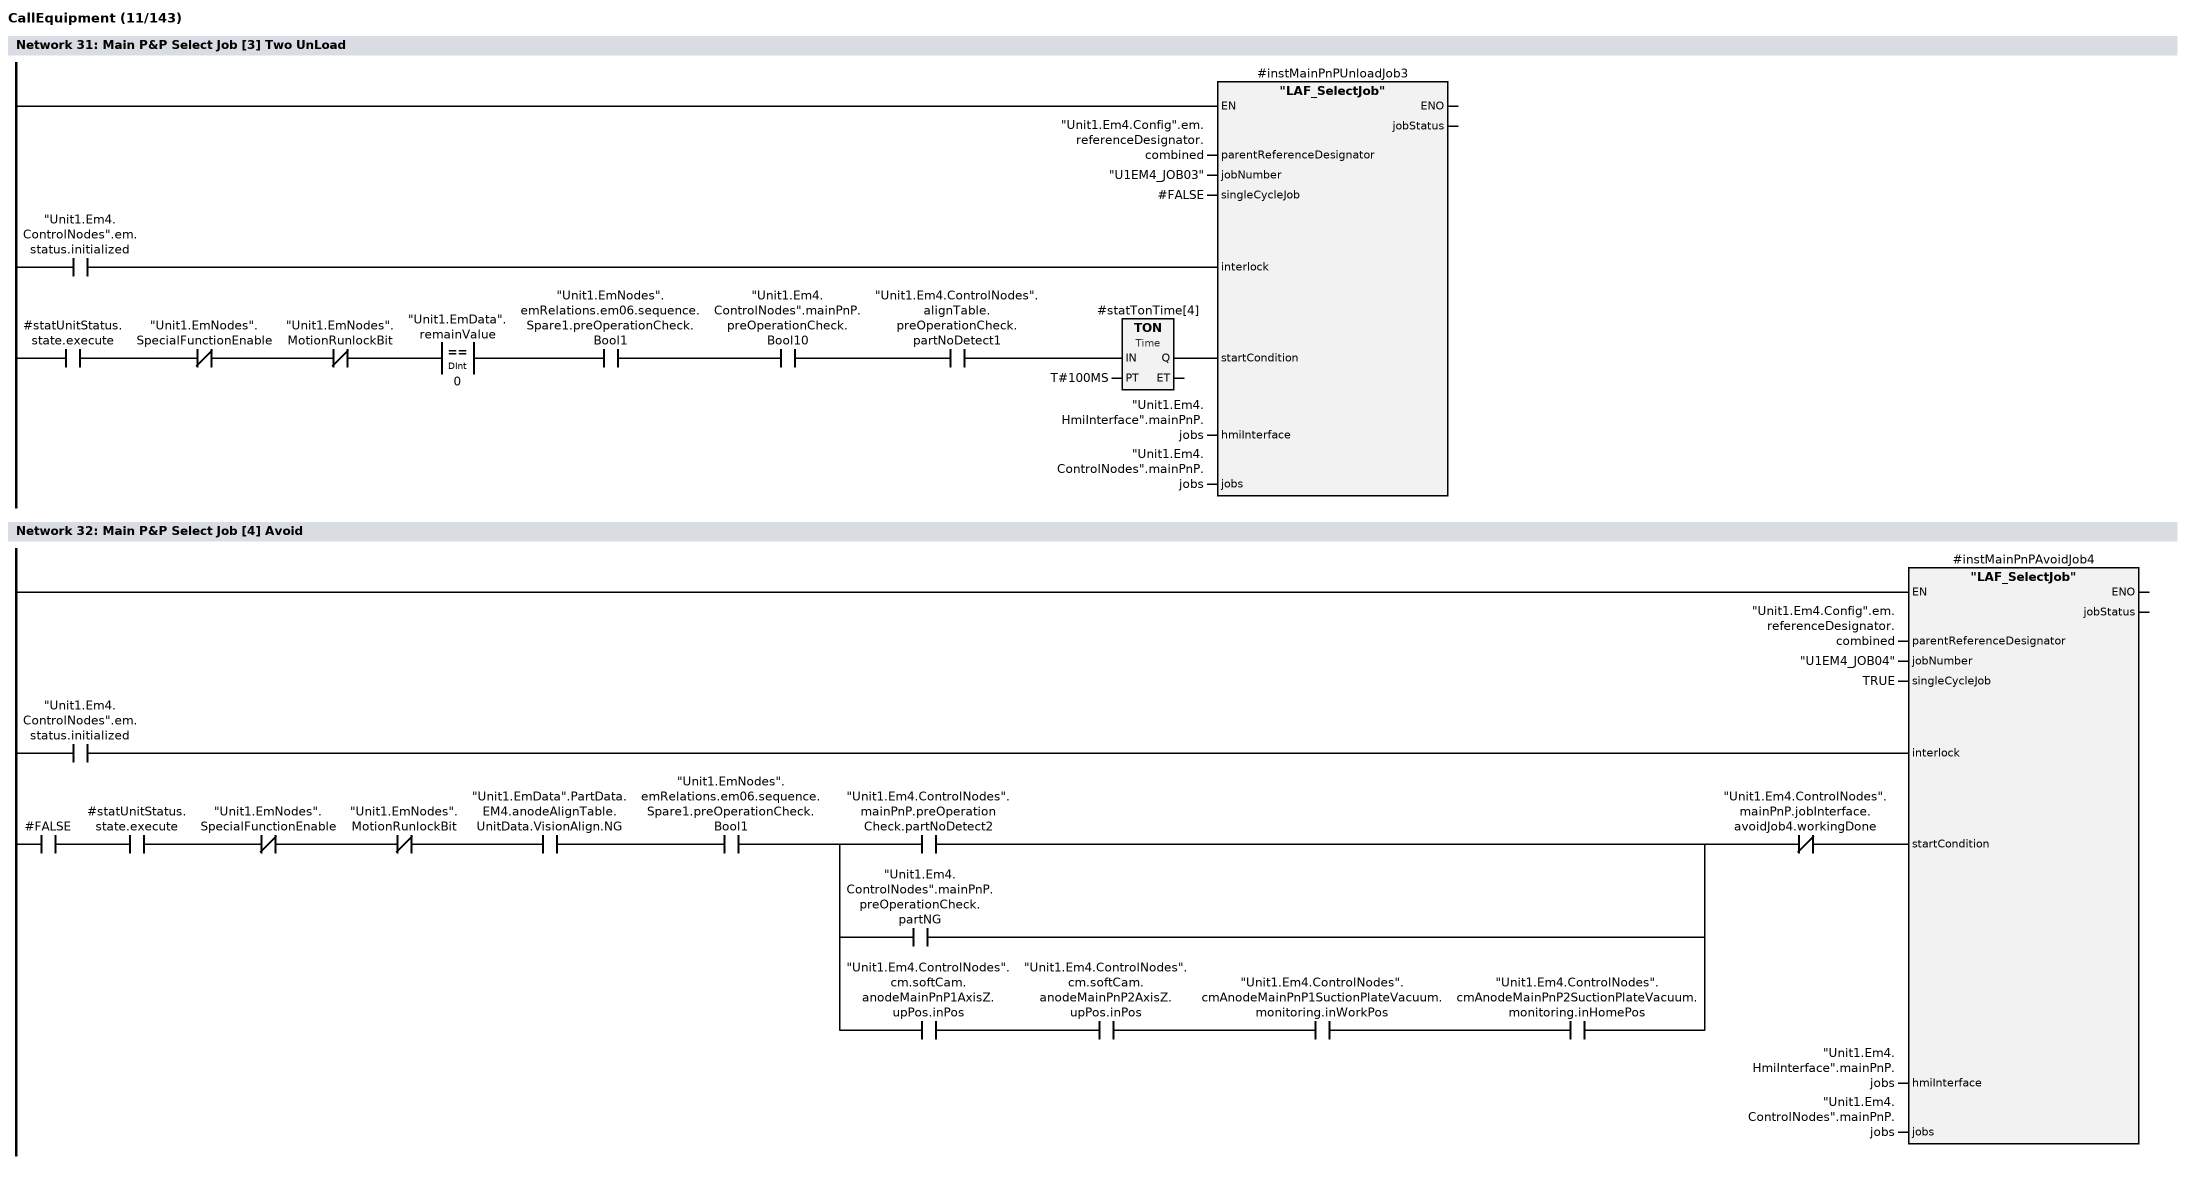
   RUNG wire#powerrail
      #instMainPnPUnloadJob3(interlock := wire#w1, startCondition := wire#w2, parentReferenceDesignator := "Unit1.Em4.Config".em.referenceDesignator.combined, jobNumber := "U1EM4_JOB03", singleCycleJob := #FALSE, hmiInterface := "Unit1.Em4.HmiInterface".mainPnP.jobs, jobs := "Unit1.Em4.ControlNodes".mainPnP.jobs, jobStatus =>)
   END_RUNG
   RUNG wire#powerrail
      Contact( "Unit1.Em4.ControlNodes".em.status.initialized )
   END_RUNG wire#w1
   RUNG wire#powerrail
      Contact( #statUnitStatus.state.execute )
      I_Contact( "Unit1.EmNodes".SpecialFunctionEnable )
      I_Contact( "Unit1.EmNodes".MotionRunlockBit )
      { S7_Templates := "SrcType := DInt" } EQ_Contact(in1 := "Unit1.EmData".remainValue, in2 := 0)
      Contact( "Unit1.EmNodes".emRelations.em06.sequence.Spare1.preOperationCheck.Bool1 )
      Contact( "Unit1.Em4.ControlNodes".mainPnP.preOperationCheck.Bool10 )
      Contact( "Unit1.Em4.ControlNodes".alignTable.preOperationCheck.partNoDetect1 )
      { S7_Templates := "time_type := Time" } #statTonTime[4].TON(pt := T#100MS, et =>)
   END_RUNG wire#w2
   // the same network as SCL:
   #statTonTime[4].TON(IN := #statUnitStatus.state.execute AND NOT "Unit1.EmNodes".SpecialFunctionEnable AND NOT "Unit1.EmNodes".MotionRunlockBit AND ("Unit1.EmData".remainValue = 0) AND "Unit1.EmNodes".emRelations.em06.sequence.Spare1.preOperationCheck.Bool1 AND "Unit1.Em4.ControlNodes".mainPnP.preOperationCheck.Bool10 AND "Unit1.Em4.ControlNodes".alignTable.preOperationCheck.partNoDetect1,
                       PT := T#100MS);
   #instMainPnPUnloadJob3(parentReferenceDesignator := "Unit1.Em4.Config".em.referenceDesignator.combined,   // "LAF_SelectJob"
                          jobNumber := "U1EM4_JOB03",
                          singleCycleJob := #FALSE,
                          interlock := "Unit1.Em4.ControlNodes".em.status.initialized,
                          startCondition := #statTonTime[4].Q,
                          hmiInterface := "Unit1.Em4.HmiInterface".mainPnP.jobs,
                          jobs := "Unit1.Em4.ControlNodes".mainPnP.jobs);
END_REGION

REGION Network 32: Main P&P Select Job [4] Avoid
   RUNG wire#powerrail
      #instMainPnPAvoidJob4(interlock := wire#w1, startCondition := wire#w4, parentReferenceDesignator := "Unit1.Em4.Config".em.referenceDesignator.combined, jobNumber := "U1EM4_JOB04", singleCycleJob := TRUE, hmiInterface := "Unit1.Em4.HmiInterface".mainPnP.jobs, jobs := "Unit1.Em4.ControlNodes".mainPnP.jobs, jobStatus =>)
   END_RUNG
   RUNG wire#powerrail
      Contact( "Unit1.Em4.ControlNodes".em.status.initialized )
   END_RUNG wire#w1
   RUNG wire#powerrail
      Contact( #FALSE )
      Contact( #statUnitStatus.state.execute )
      I_Contact( "Unit1.EmNodes".SpecialFunctionEnable )
      I_Contact( "Unit1.EmNodes".MotionRunlockBit )
      Contact( "Unit1.EmData".PartData.EM4.anodeAlignTable.UnitData.VisionAlign.NG )
      Contact( "Unit1.EmNodes".emRelations.em06.sequence.Spare1.preOperationCheck.Bool1 )
      wire#w2
      Contact( "Unit1.Em4.ControlNodes".mainPnP.preOperationCheck.partNoDetect2 )
      wire#w3
      I_Contact( "Unit1.Em4.ControlNodes".mainPnP.jobInterface.avoidJob4.workingDone )
   END_RUNG wire#w4
   RUNG wire#w2
      Contact( "Unit1.Em4.ControlNodes".mainPnP.preOperationCheck.partNG )
   END_RUNG wire#w3
   RUNG wire#w2
      Contact( "Unit1.Em4.ControlNodes".cm.softCam.anodeMainPnP1AxisZ.upPos.inPos )
      Contact( "Unit1.Em4.ControlNodes".cm.softCam.anodeMainPnP2AxisZ.upPos.inPos )
      Contact( "Unit1.Em4.ControlNodes".cmAnodeMainPnP1SuctionPlateVacuum.monitoring.inWorkPos )
      Contact( "Unit1.Em4.ControlNodes".cmAnodeMainPnP2SuctionPlateVacuum.monitoring.inHomePos )
   END_RUNG wire#w3
   // the same network as SCL:
   #instMainPnPAvoidJob4(parentReferenceDesignator := "Unit1.Em4.Config".em.referenceDesignator.combined,   // "LAF_SelectJob"
                         jobNumber := "U1EM4_JOB04",
                         singleCycleJob := TRUE,
                         interlock := "Unit1.Em4.ControlNodes".em.status.initialized,
                         startCondition := #FALSE AND #statUnitStatus.state.execute AND NOT "Unit1.EmNodes".SpecialFunctionEnable AND NOT "Unit1.EmNodes".MotionRunlockBit AND "Unit1.EmData".PartData.EM4.anodeAlignTable.UnitData.VisionAlign.NG AND "Unit1.EmNodes".emRelations.em06.sequence.Spare1.preOperationCheck.Bool1 AND ("Unit1.Em4.ControlNodes".mainPnP.preOperationCheck.partNoDetect2 OR "Unit1.Em4.ControlNodes".mainPnP.preOperationCheck.partNG OR ("Unit1.Em4.ControlNodes".cm.softCam.anodeMainPnP1AxisZ.upPos.inPos AND "Unit1.Em4.ControlNodes".cm.softCam.anodeMainPnP2AxisZ.upPos.inPos AND "Unit1.Em4.ControlNodes".cmAnodeMainPnP1SuctionPlateVacuum.monitoring.inWorkPos AND "Unit1.Em4.ControlNodes".cmAnodeMainPnP2SuctionPlateVacuum.monitoring.inHomePos)) AND NOT "Unit1.Em4.ControlNodes".mainPnP.jobInterface.avoidJob4.workingDone,
                         hmiInterface := "Unit1.Em4.HmiInterface".mainPnP.jobs,
                         jobs := "Unit1.Em4.ControlNodes".mainPnP.jobs);
END_REGION

REGION Network 33: Main P&P Select Job [7] Down Gripper Wait
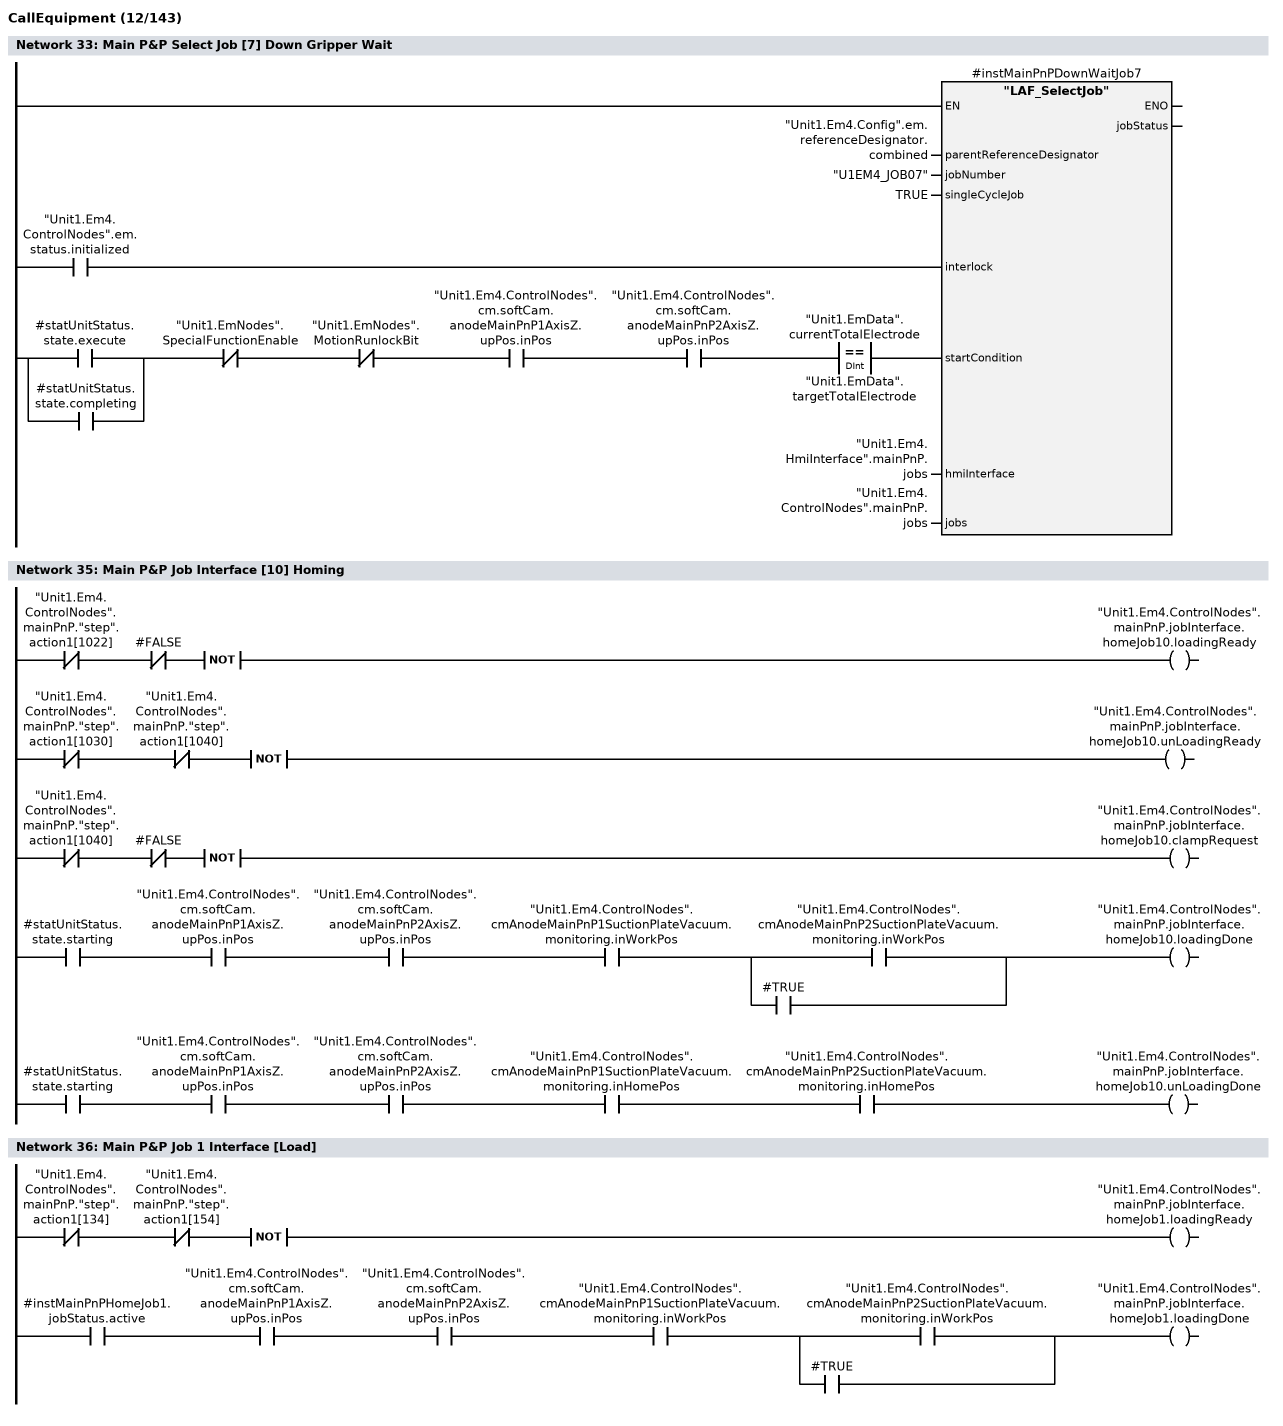
   RUNG wire#powerrail
      #instMainPnPDownWaitJob7(interlock := wire#w1, startCondition := wire#w3, parentReferenceDesignator := "Unit1.Em4.Config".em.referenceDesignator.combined, jobNumber := "U1EM4_JOB07", singleCycleJob := TRUE, hmiInterface := "Unit1.Em4.HmiInterface".mainPnP.jobs, jobs := "Unit1.Em4.ControlNodes".mainPnP.jobs, jobStatus =>)
   END_RUNG
   RUNG wire#powerrail
      Contact( "Unit1.Em4.ControlNodes".em.status.initialized )
   END_RUNG wire#w1
   RUNG wire#powerrail
      Contact( #statUnitStatus.state.execute )
      wire#w2
      I_Contact( "Unit1.EmNodes".SpecialFunctionEnable )
      I_Contact( "Unit1.EmNodes".MotionRunlockBit )
      Contact( "Unit1.Em4.ControlNodes".cm.softCam.anodeMainPnP1AxisZ.upPos.inPos )
      Contact( "Unit1.Em4.ControlNodes".cm.softCam.anodeMainPnP2AxisZ.upPos.inPos )
      { S7_Templates := "SrcType := DInt" } EQ_Contact(in1 := "Unit1.EmData".currentTotalElectrode, in2 := "Unit1.EmData".targetTotalElectrode)
   END_RUNG wire#w3
   RUNG wire#powerrail
      Contact( #statUnitStatus.state.completing )
   END_RUNG wire#w2
   // the same network as SCL:
   #instMainPnPDownWaitJob7(parentReferenceDesignator := "Unit1.Em4.Config".em.referenceDesignator.combined,   // "LAF_SelectJob"
                           jobNumber := "U1EM4_JOB07",
                           singleCycleJob := TRUE,
                           interlock := "Unit1.Em4.ControlNodes".em.status.initialized,
                           startCondition := (#statUnitStatus.state.execute OR #statUnitStatus.state.completing) AND NOT "Unit1.EmNodes".SpecialFunctionEnable AND NOT "Unit1.EmNodes".MotionRunlockBit AND "Unit1.Em4.ControlNodes".cm.softCam.anodeMainPnP1AxisZ.upPos.inPos AND "Unit1.Em4.ControlNodes".cm.softCam.anodeMainPnP2AxisZ.upPos.inPos AND ("Unit1.EmData".currentTotalElectrode = "Unit1.EmData".targetTotalElectrode),
                           hmiInterface := "Unit1.Em4.HmiInterface".mainPnP.jobs,
                           jobs := "Unit1.Em4.ControlNodes".mainPnP.jobs);
END_REGION

REGION Network 35: Main P&P Job Interface [10] Homing
   RUNG wire#powerrail
      I_Contact( "Unit1.Em4.ControlNodes".mainPnP."step".action1[1022] )
      I_Contact( #FALSE )
      Not()
      Coil( "Unit1.Em4.ControlNodes".mainPnP.jobInterface.homeJob10.loadingReady )
   END_RUNG
   RUNG wire#powerrail
      I_Contact( "Unit1.Em4.ControlNodes".mainPnP."step".action1[1030] )
      I_Contact( "Unit1.Em4.ControlNodes".mainPnP."step".action1[1040] )
      Not()
      Coil( "Unit1.Em4.ControlNodes".mainPnP.jobInterface.homeJob10.unLoadingReady )
   END_RUNG
   RUNG wire#powerrail
      I_Contact( "Unit1.Em4.ControlNodes".mainPnP."step".action1[1040] )
      I_Contact( #FALSE )
      Not()
      Coil( "Unit1.Em4.ControlNodes".mainPnP.jobInterface.homeJob10.clampRequest )
   END_RUNG
   RUNG wire#powerrail
      Contact( #statUnitStatus.state.starting )
      Contact( "Unit1.Em4.ControlNodes".cm.softCam.anodeMainPnP1AxisZ.upPos.inPos )
      Contact( "Unit1.Em4.ControlNodes".cm.softCam.anodeMainPnP2AxisZ.upPos.inPos )
      Contact( "Unit1.Em4.ControlNodes".cmAnodeMainPnP1SuctionPlateVacuum.monitoring.inWorkPos )
      wire#w1
      Contact( "Unit1.Em4.ControlNodes".cmAnodeMainPnP2SuctionPlateVacuum.monitoring.inWorkPos )
      wire#w2
      Coil( "Unit1.Em4.ControlNodes".mainPnP.jobInterface.homeJob10.loadingDone )
   END_RUNG
   RUNG wire#w1
      Contact( #TRUE )
   END_RUNG wire#w2
   RUNG wire#powerrail
      Contact( #statUnitStatus.state.starting )
      Contact( "Unit1.Em4.ControlNodes".cm.softCam.anodeMainPnP1AxisZ.upPos.inPos )
      Contact( "Unit1.Em4.ControlNodes".cm.softCam.anodeMainPnP2AxisZ.upPos.inPos )
      Contact( "Unit1.Em4.ControlNodes".cmAnodeMainPnP1SuctionPlateVacuum.monitoring.inHomePos )
      Contact( "Unit1.Em4.ControlNodes".cmAnodeMainPnP2SuctionPlateVacuum.monitoring.inHomePos )
      Coil( "Unit1.Em4.ControlNodes".mainPnP.jobInterface.homeJob10.unLoadingDone )
   END_RUNG
   // the same network as SCL:
   "Unit1.Em4.ControlNodes".mainPnP.jobInterface.homeJob10.loadingReady := NOT (NOT "Unit1.Em4.ControlNodes".mainPnP."step".action1[1022] AND NOT #FALSE);
   "Unit1.Em4.ControlNodes".mainPnP.jobInterface.homeJob10.unLoadingReady := NOT (NOT "Unit1.Em4.ControlNodes".mainPnP."step".action1[1030] AND NOT "Unit1.Em4.ControlNodes".mainPnP."step".action1[1040]);
   "Unit1.Em4.ControlNodes".mainPnP.jobInterface.homeJob10.clampRequest := NOT (NOT "Unit1.Em4.ControlNodes".mainPnP."step".action1[1040] AND NOT #FALSE);
   "Unit1.Em4.ControlNodes".mainPnP.jobInterface.homeJob10.loadingDone := #statUnitStatus.state.starting AND "Unit1.Em4.ControlNodes".cm.softCam.anodeMainPnP1AxisZ.upPos.inPos AND "Unit1.Em4.ControlNodes".cm.softCam.anodeMainPnP2AxisZ.upPos.inPos AND "Unit1.Em4.ControlNodes".cmAnodeMainPnP1SuctionPlateVacuum.monitoring.inWorkPos AND ("Unit1.Em4.ControlNodes".cmAnodeMainPnP2SuctionPlateVacuum.monitoring.inWorkPos OR #TRUE);
   "Unit1.Em4.ControlNodes".mainPnP.jobInterface.homeJob10.unLoadingDone := #statUnitStatus.state.starting AND "Unit1.Em4.ControlNodes".cm.softCam.anodeMainPnP1AxisZ.upPos.inPos AND "Unit1.Em4.ControlNodes".cm.softCam.anodeMainPnP2AxisZ.upPos.inPos AND "Unit1.Em4.ControlNodes".cmAnodeMainPnP1SuctionPlateVacuum.monitoring.inHomePos AND "Unit1.Em4.ControlNodes".cmAnodeMainPnP2SuctionPlateVacuum.monitoring.inHomePos;
END_REGION

REGION Network 36: Main P&P Job 1 Interface [Load]
   RUNG wire#powerrail
      I_Contact( "Unit1.Em4.ControlNodes".mainPnP."step".action1[134] )
      I_Contact( "Unit1.Em4.ControlNodes".mainPnP."step".action1[154] )
      Not()
      Coil( "Unit1.Em4.ControlNodes".mainPnP.jobInterface.homeJob1.loadingReady )
   END_RUNG
   RUNG wire#powerrail
      Contact( #instMainPnPHomeJob1.jobStatus.active )
      Contact( "Unit1.Em4.ControlNodes".cm.softCam.anodeMainPnP1AxisZ.upPos.inPos )
      Contact( "Unit1.Em4.ControlNodes".cm.softCam.anodeMainPnP2AxisZ.upPos.inPos )
      Contact( "Unit1.Em4.ControlNodes".cmAnodeMainPnP1SuctionPlateVacuum.monitoring.inWorkPos )
      wire#w1
      Contact( "Unit1.Em4.ControlNodes".cmAnodeMainPnP2SuctionPlateVacuum.monitoring.inWorkPos )
      wire#w2
      Coil( "Unit1.Em4.ControlNodes".mainPnP.jobInterface.homeJob1.loadingDone )
   END_RUNG
   RUNG wire#w1
      Contact( #TRUE )
   END_RUNG wire#w2
   // the same network as SCL:
   "Unit1.Em4.ControlNodes".mainPnP.jobInterface.homeJob1.loadingReady := NOT (NOT "Unit1.Em4.ControlNodes".mainPnP."step".action1[134] AND NOT "Unit1.Em4.ControlNodes".mainPnP."step".action1[154]);
   "Unit1.Em4.ControlNodes".mainPnP.jobInterface.homeJob1.loadingDone := #instMainPnPHomeJob1.jobStatus.active AND "Unit1.Em4.ControlNodes".cm.softCam.anodeMainPnP1AxisZ.upPos.inPos AND "Unit1.Em4.ControlNodes".cm.softCam.anodeMainPnP2AxisZ.upPos.inPos AND "Unit1.Em4.ControlNodes".cmAnodeMainPnP1SuctionPlateVacuum.monitoring.inWorkPos AND ("Unit1.Em4.ControlNodes".cmAnodeMainPnP2SuctionPlateVacuum.monitoring.inWorkPos OR #TRUE);
END_REGION

REGION Network 37: Main P&P Job 1 Interface [Unload]
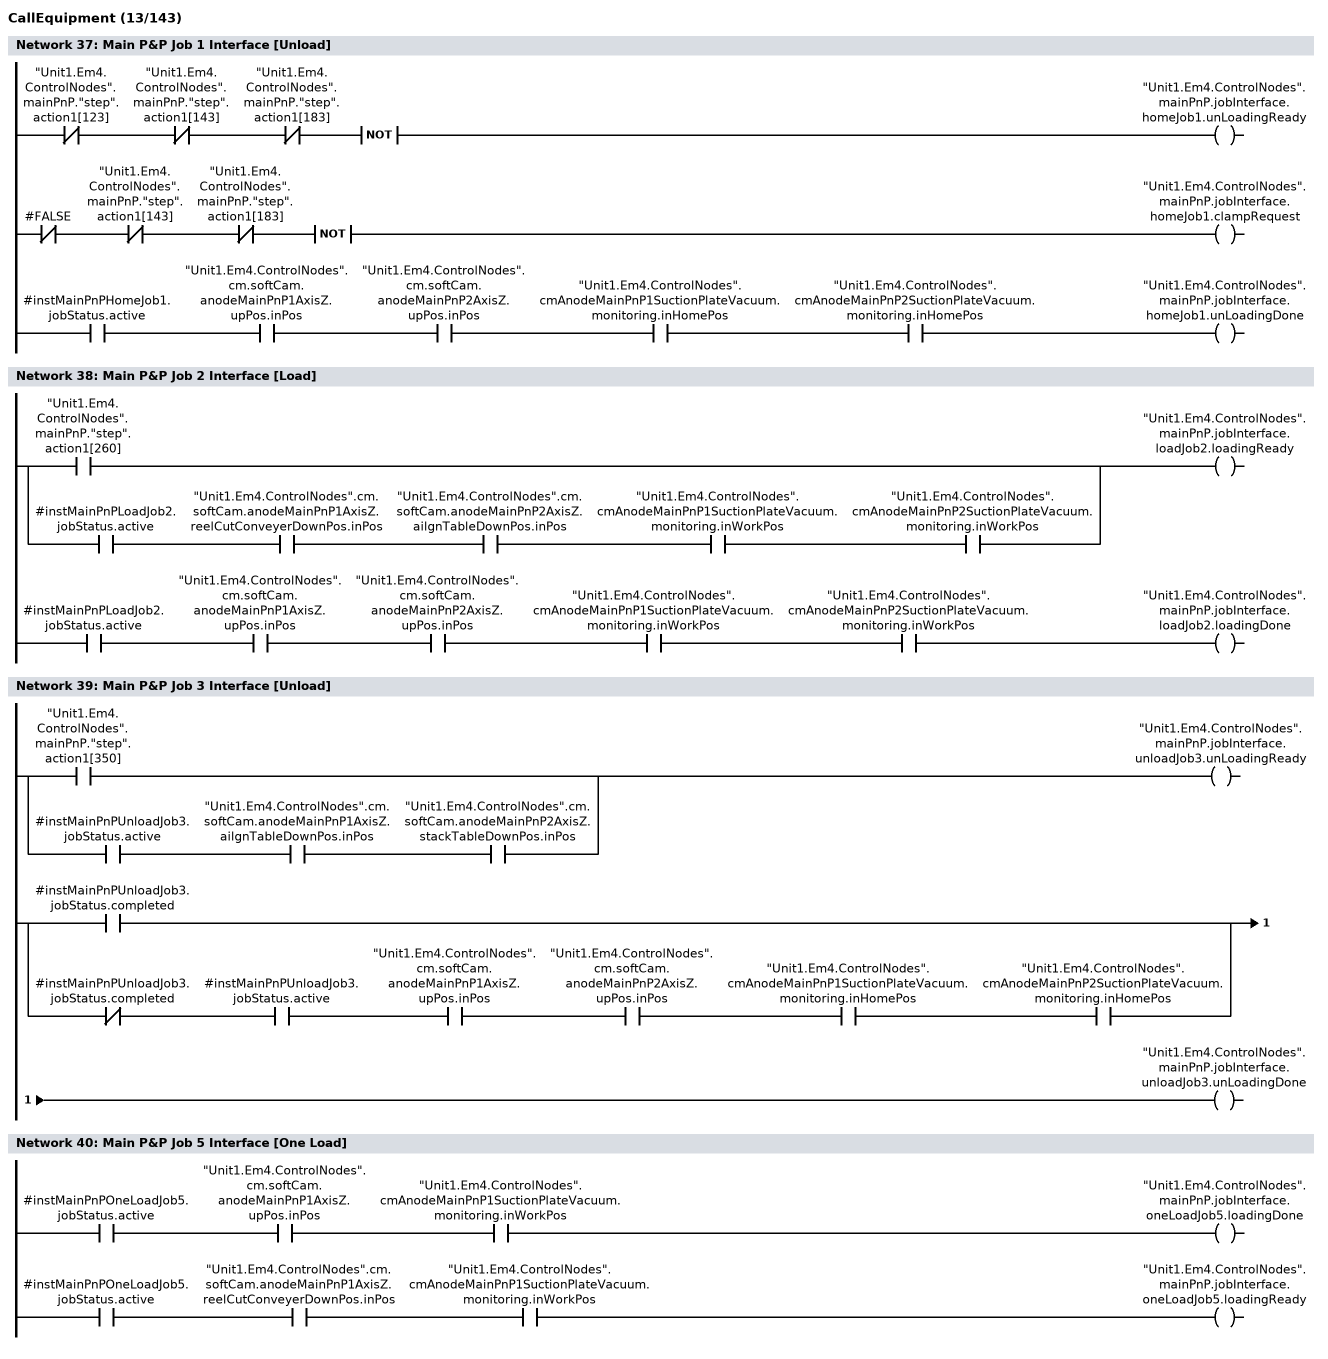
   RUNG wire#powerrail
      I_Contact( "Unit1.Em4.ControlNodes".mainPnP."step".action1[123] )
      I_Contact( "Unit1.Em4.ControlNodes".mainPnP."step".action1[143] )
      I_Contact( "Unit1.Em4.ControlNodes".mainPnP."step".action1[183] )
      Not()
      Coil( "Unit1.Em4.ControlNodes".mainPnP.jobInterface.homeJob1.unLoadingReady )
   END_RUNG
   RUNG wire#powerrail
      I_Contact( #FALSE )
      I_Contact( "Unit1.Em4.ControlNodes".mainPnP."step".action1[143] )
      I_Contact( "Unit1.Em4.ControlNodes".mainPnP."step".action1[183] )
      Not()
      Coil( "Unit1.Em4.ControlNodes".mainPnP.jobInterface.homeJob1.clampRequest )
   END_RUNG
   RUNG wire#powerrail
      Contact( #instMainPnPHomeJob1.jobStatus.active )
      Contact( "Unit1.Em4.ControlNodes".cm.softCam.anodeMainPnP1AxisZ.upPos.inPos )
      Contact( "Unit1.Em4.ControlNodes".cm.softCam.anodeMainPnP2AxisZ.upPos.inPos )
      Contact( "Unit1.Em4.ControlNodes".cmAnodeMainPnP1SuctionPlateVacuum.monitoring.inHomePos )
      Contact( "Unit1.Em4.ControlNodes".cmAnodeMainPnP2SuctionPlateVacuum.monitoring.inHomePos )
      Coil( "Unit1.Em4.ControlNodes".mainPnP.jobInterface.homeJob1.unLoadingDone )
   END_RUNG
   // the same network as SCL:
   "Unit1.Em4.ControlNodes".mainPnP.jobInterface.homeJob1.unLoadingReady := NOT (NOT "Unit1.Em4.ControlNodes".mainPnP."step".action1[123] AND NOT "Unit1.Em4.ControlNodes".mainPnP."step".action1[143] AND NOT "Unit1.Em4.ControlNodes".mainPnP."step".action1[183]);
   "Unit1.Em4.ControlNodes".mainPnP.jobInterface.homeJob1.clampRequest := NOT (NOT #FALSE AND NOT "Unit1.Em4.ControlNodes".mainPnP."step".action1[143] AND NOT "Unit1.Em4.ControlNodes".mainPnP."step".action1[183]);
   "Unit1.Em4.ControlNodes".mainPnP.jobInterface.homeJob1.unLoadingDone := #instMainPnPHomeJob1.jobStatus.active AND "Unit1.Em4.ControlNodes".cm.softCam.anodeMainPnP1AxisZ.upPos.inPos AND "Unit1.Em4.ControlNodes".cm.softCam.anodeMainPnP2AxisZ.upPos.inPos AND "Unit1.Em4.ControlNodes".cmAnodeMainPnP1SuctionPlateVacuum.monitoring.inHomePos AND "Unit1.Em4.ControlNodes".cmAnodeMainPnP2SuctionPlateVacuum.monitoring.inHomePos;
END_REGION

REGION Network 38: Main P&P Job 2 Interface [Load]
   RUNG wire#powerrail
      Contact( "Unit1.Em4.ControlNodes".mainPnP."step".action1[260] )
      wire#w1
      Coil( "Unit1.Em4.ControlNodes".mainPnP.jobInterface.loadJob2.loadingReady )
   END_RUNG
   RUNG wire#powerrail
      Contact( #instMainPnPLoadJob2.jobStatus.active )
      Contact( "Unit1.Em4.ControlNodes".cm.softCam.anodeMainPnP1AxisZ.reelCutConveyerDownPos.inPos )
      Contact( "Unit1.Em4.ControlNodes".cm.softCam.anodeMainPnP2AxisZ.ailgnTableDownPos.inPos )
      Contact( "Unit1.Em4.ControlNodes".cmAnodeMainPnP1SuctionPlateVacuum.monitoring.inWorkPos )
      Contact( "Unit1.Em4.ControlNodes".cmAnodeMainPnP2SuctionPlateVacuum.monitoring.inWorkPos )
   END_RUNG wire#w1
   RUNG wire#powerrail
      Contact( #instMainPnPLoadJob2.jobStatus.active )
      Contact( "Unit1.Em4.ControlNodes".cm.softCam.anodeMainPnP1AxisZ.upPos.inPos )
      Contact( "Unit1.Em4.ControlNodes".cm.softCam.anodeMainPnP2AxisZ.upPos.inPos )
      Contact( "Unit1.Em4.ControlNodes".cmAnodeMainPnP1SuctionPlateVacuum.monitoring.inWorkPos )
      Contact( "Unit1.Em4.ControlNodes".cmAnodeMainPnP2SuctionPlateVacuum.monitoring.inWorkPos )
      Coil( "Unit1.Em4.ControlNodes".mainPnP.jobInterface.loadJob2.loadingDone )
   END_RUNG
   // the same network as SCL:
   "Unit1.Em4.ControlNodes".mainPnP.jobInterface.loadJob2.loadingReady := "Unit1.Em4.ControlNodes".mainPnP."step".action1[260] OR (#instMainPnPLoadJob2.jobStatus.active AND "Unit1.Em4.ControlNodes".cm.softCam.anodeMainPnP1AxisZ.reelCutConveyerDownPos.inPos AND "Unit1.Em4.ControlNodes".cm.softCam.anodeMainPnP2AxisZ.ailgnTableDownPos.inPos AND "Unit1.Em4.ControlNodes".cmAnodeMainPnP1SuctionPlateVacuum.monitoring.inWorkPos AND "Unit1.Em4.ControlNodes".cmAnodeMainPnP2SuctionPlateVacuum.monitoring.inWorkPos);
   "Unit1.Em4.ControlNodes".mainPnP.jobInterface.loadJob2.loadingDone := #instMainPnPLoadJob2.jobStatus.active AND "Unit1.Em4.ControlNodes".cm.softCam.anodeMainPnP1AxisZ.upPos.inPos AND "Unit1.Em4.ControlNodes".cm.softCam.anodeMainPnP2AxisZ.upPos.inPos AND "Unit1.Em4.ControlNodes".cmAnodeMainPnP1SuctionPlateVacuum.monitoring.inWorkPos AND "Unit1.Em4.ControlNodes".cmAnodeMainPnP2SuctionPlateVacuum.monitoring.inWorkPos;
END_REGION

REGION Network 39: Main P&P Job 3 Interface [Unload]
   RUNG wire#powerrail
      Contact( "Unit1.Em4.ControlNodes".mainPnP."step".action1[350] )
      wire#w1
      Coil( "Unit1.Em4.ControlNodes".mainPnP.jobInterface.unloadJob3.unLoadingReady )
   END_RUNG
   RUNG wire#powerrail
      Contact( #instMainPnPUnloadJob3.jobStatus.active )
      Contact( "Unit1.Em4.ControlNodes".cm.softCam.anodeMainPnP1AxisZ.ailgnTableDownPos.inPos )
      Contact( "Unit1.Em4.ControlNodes".cm.softCam.anodeMainPnP2AxisZ.stackTableDownPos.inPos )
   END_RUNG wire#w1
   RUNG wire#powerrail
      Contact( #instMainPnPUnloadJob3.jobStatus.completed )
      wire#w2
      Coil( "Unit1.Em4.ControlNodes".mainPnP.jobInterface.unloadJob3.unLoadingDone )
   END_RUNG
   RUNG wire#powerrail
      I_Contact( #instMainPnPUnloadJob3.jobStatus.completed )
      Contact( #instMainPnPUnloadJob3.jobStatus.active )
      Contact( "Unit1.Em4.ControlNodes".cm.softCam.anodeMainPnP1AxisZ.upPos.inPos )
      Contact( "Unit1.Em4.ControlNodes".cm.softCam.anodeMainPnP2AxisZ.upPos.inPos )
      Contact( "Unit1.Em4.ControlNodes".cmAnodeMainPnP1SuctionPlateVacuum.monitoring.inHomePos )
      Contact( "Unit1.Em4.ControlNodes".cmAnodeMainPnP2SuctionPlateVacuum.monitoring.inHomePos )
   END_RUNG wire#w2
   // the same network as SCL:
   "Unit1.Em4.ControlNodes".mainPnP.jobInterface.unloadJob3.unLoadingReady := "Unit1.Em4.ControlNodes".mainPnP."step".action1[350] OR (#instMainPnPUnloadJob3.jobStatus.active AND "Unit1.Em4.ControlNodes".cm.softCam.anodeMainPnP1AxisZ.ailgnTableDownPos.inPos AND "Unit1.Em4.ControlNodes".cm.softCam.anodeMainPnP2AxisZ.stackTableDownPos.inPos);
   "Unit1.Em4.ControlNodes".mainPnP.jobInterface.unloadJob3.unLoadingDone := #instMainPnPUnloadJob3.jobStatus.completed OR (NOT #instMainPnPUnloadJob3.jobStatus.completed AND #instMainPnPUnloadJob3.jobStatus.active AND "Unit1.Em4.ControlNodes".cm.softCam.anodeMainPnP1AxisZ.upPos.inPos AND "Unit1.Em4.ControlNodes".cm.softCam.anodeMainPnP2AxisZ.upPos.inPos AND "Unit1.Em4.ControlNodes".cmAnodeMainPnP1SuctionPlateVacuum.monitoring.inHomePos AND "Unit1.Em4.ControlNodes".cmAnodeMainPnP2SuctionPlateVacuum.monitoring.inHomePos);
END_REGION

REGION Network 40: Main P&P Job 5 Interface [One Load]
   RUNG wire#powerrail
      Contact( #instMainPnPOneLoadJob5.jobStatus.active )
      Contact( "Unit1.Em4.ControlNodes".cm.softCam.anodeMainPnP1AxisZ.upPos.inPos )
      Contact( "Unit1.Em4.ControlNodes".cmAnodeMainPnP1SuctionPlateVacuum.monitoring.inWorkPos )
      Coil( "Unit1.Em4.ControlNodes".mainPnP.jobInterface.oneLoadJob5.loadingDone )
   END_RUNG
   RUNG wire#powerrail
      Contact( #instMainPnPOneLoadJob5.jobStatus.active )
      Contact( "Unit1.Em4.ControlNodes".cm.softCam.anodeMainPnP1AxisZ.reelCutConveyerDownPos.inPos )
      Contact( "Unit1.Em4.ControlNodes".cmAnodeMainPnP1SuctionPlateVacuum.monitoring.inWorkPos )
      Coil( "Unit1.Em4.ControlNodes".mainPnP.jobInterface.oneLoadJob5.loadingReady )
   END_RUNG
   // the same network as SCL:
   "Unit1.Em4.ControlNodes".mainPnP.jobInterface.oneLoadJob5.loadingDone := #instMainPnPOneLoadJob5.jobStatus.active AND "Unit1.Em4.ControlNodes".cm.softCam.anodeMainPnP1AxisZ.upPos.inPos AND "Unit1.Em4.ControlNodes".cmAnodeMainPnP1SuctionPlateVacuum.monitoring.inWorkPos;
   "Unit1.Em4.ControlNodes".mainPnP.jobInterface.oneLoadJob5.loadingReady := #instMainPnPOneLoadJob5.jobStatus.active AND "Unit1.Em4.ControlNodes".cm.softCam.anodeMainPnP1AxisZ.reelCutConveyerDownPos.inPos AND "Unit1.Em4.ControlNodes".cmAnodeMainPnP1SuctionPlateVacuum.monitoring.inWorkPos;
END_REGION

REGION Network 41: Main P&P Job 6 Interface [One Unload]
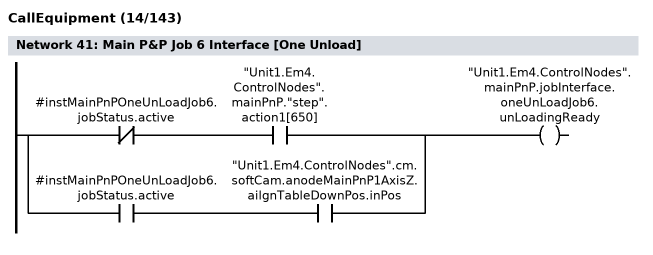
   RUNG wire#powerrail
      I_Contact( #instMainPnPOneUnLoadJob6.jobStatus.active )
      Contact( "Unit1.Em4.ControlNodes".mainPnP."step".action1[650] )
      wire#w1
      Coil( "Unit1.Em4.ControlNodes".mainPnP.jobInterface.oneUnLoadJob6.unLoadingReady )
   END_RUNG
   RUNG wire#powerrail
      Contact( #instMainPnPOneUnLoadJob6.jobStatus.active )
      Contact( "Unit1.Em4.ControlNodes".cm.softCam.anodeMainPnP1AxisZ.ailgnTableDownPos.inPos )
   END_RUNG wire#w1
   // the same network as SCL:
   "Unit1.Em4.ControlNodes".mainPnP.jobInterface.oneUnLoadJob6.unLoadingReady := (NOT #instMainPnPOneUnLoadJob6.jobStatus.active AND "Unit1.Em4.ControlNodes".mainPnP."step".action1[650]) OR (#instMainPnPOneUnLoadJob6.jobStatus.active AND "Unit1.Em4.ControlNodes".cm.softCam.anodeMainPnP1AxisZ.ailgnTableDownPos.inPos);
END_REGION

REGION Network 42: Main P&P Job Interface Working Done
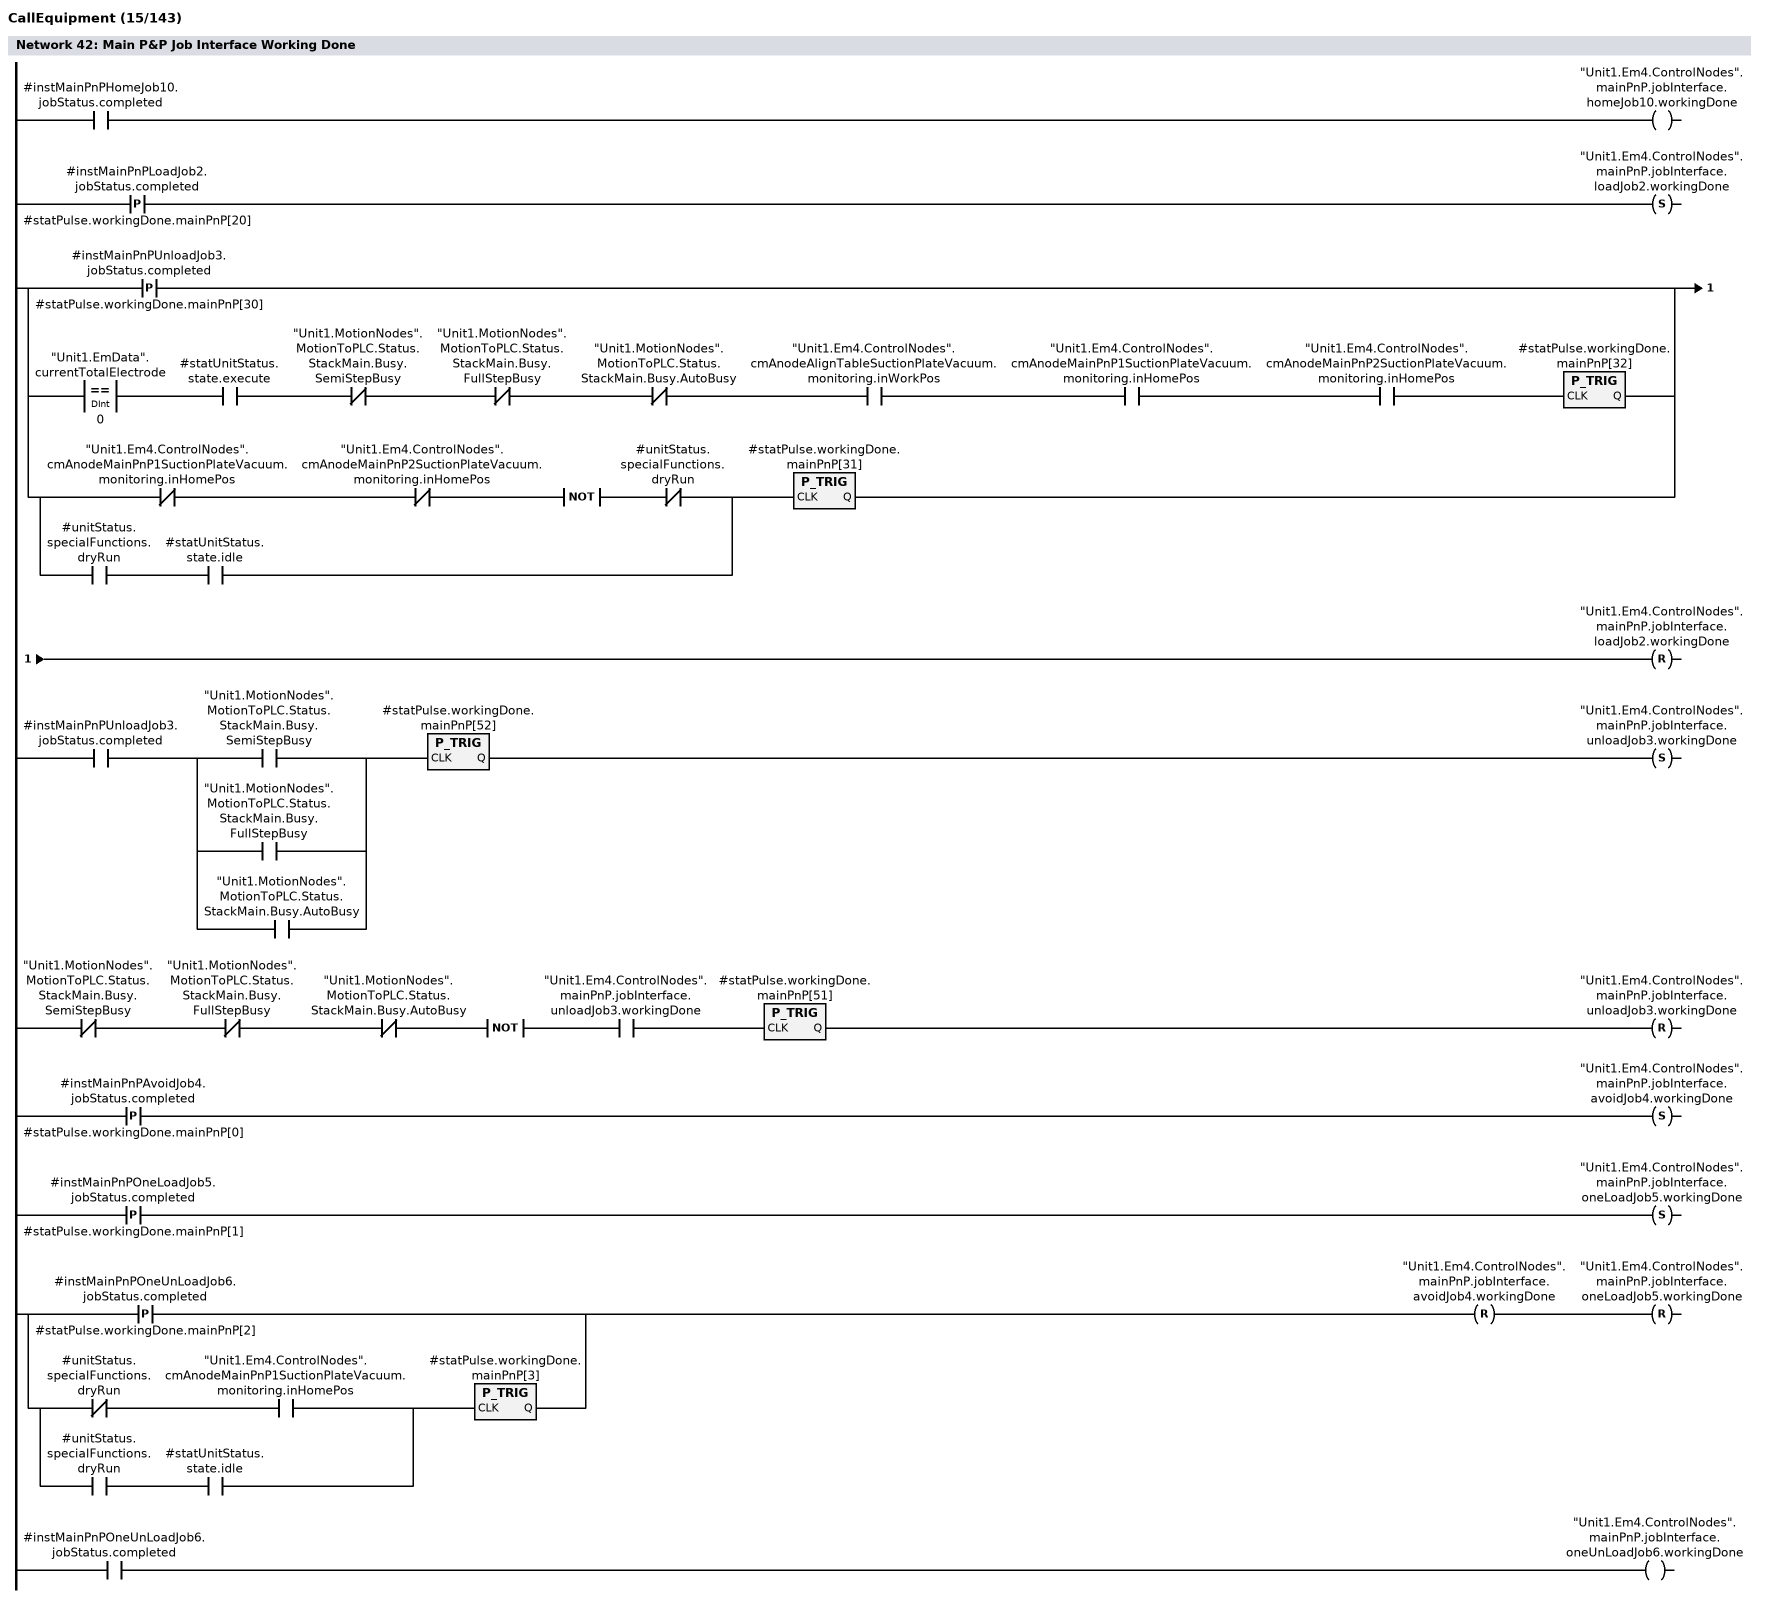
   RUNG wire#powerrail
      Contact( #instMainPnPHomeJob10.jobStatus.completed )
      Coil( "Unit1.Em4.ControlNodes".mainPnP.jobInterface.homeJob10.workingDone )
   END_RUNG
   RUNG wire#powerrail
      P_Contact(operand := #instMainPnPLoadJob2.jobStatus.completed, bit := #statPulse.workingDone.mainPnP[20])
      S_Coil( "Unit1.Em4.ControlNodes".mainPnP.jobInterface.loadJob2.workingDone )
   END_RUNG
   RUNG wire#powerrail
      P_Contact(operand := #instMainPnPUnloadJob3.jobStatus.completed, bit := #statPulse.workingDone.mainPnP[30])
      wire#w1
      R_Coil( "Unit1.Em4.ControlNodes".mainPnP.jobInterface.loadJob2.workingDone )
   END_RUNG
   RUNG wire#powerrail
      { S7_Templates := "SrcType := DInt" } EQ_Contact(in1 := "Unit1.EmData".currentTotalElectrode, in2 := 0)
      Contact( #statUnitStatus.state.execute )
      I_Contact( "Unit1.MotionNodes".MotionToPLC.Status.StackMain.Busy.SemiStepBusy )
      I_Contact( "Unit1.MotionNodes".MotionToPLC.Status.StackMain.Busy.FullStepBusy )
      I_Contact( "Unit1.MotionNodes".MotionToPLC.Status.StackMain.Busy.AutoBusy )
      Contact( "Unit1.Em4.ControlNodes".cmAnodeAlignTableSuctionPlateVacuum.monitoring.inWorkPos )
      Contact( "Unit1.Em4.ControlNodes".cmAnodeMainPnP1SuctionPlateVacuum.monitoring.inHomePos )
      Contact( "Unit1.Em4.ControlNodes".cmAnodeMainPnP2SuctionPlateVacuum.monitoring.inHomePos )
      P_Trig( #statPulse.workingDone.mainPnP[32] )
   END_RUNG wire#w1
   RUNG wire#powerrail
      I_Contact( "Unit1.Em4.ControlNodes".cmAnodeMainPnP1SuctionPlateVacuum.monitoring.inHomePos )
      I_Contact( "Unit1.Em4.ControlNodes".cmAnodeMainPnP2SuctionPlateVacuum.monitoring.inHomePos )
      Not()
      I_Contact( #unitStatus.specialFunctions.dryRun )
      wire#w2
      P_Trig( #statPulse.workingDone.mainPnP[31] )
   END_RUNG wire#w1
   RUNG wire#powerrail
      Contact( #unitStatus.specialFunctions.dryRun )
      Contact( #statUnitStatus.state.idle )
   END_RUNG wire#w2
   RUNG wire#powerrail
      Contact( #instMainPnPUnloadJob3.jobStatus.completed )
      wire#w3
      Contact( "Unit1.MotionNodes".MotionToPLC.Status.StackMain.Busy.SemiStepBusy )
      wire#w4
      P_Trig( #statPulse.workingDone.mainPnP[52] )
      S_Coil( "Unit1.Em4.ControlNodes".mainPnP.jobInterface.unloadJob3.workingDone )
   END_RUNG
   RUNG wire#w3
      Contact( "Unit1.MotionNodes".MotionToPLC.Status.StackMain.Busy.FullStepBusy )
   END_RUNG wire#w4
   RUNG wire#w3
      Contact( "Unit1.MotionNodes".MotionToPLC.Status.StackMain.Busy.AutoBusy )
   END_RUNG wire#w4
   RUNG wire#powerrail
      I_Contact( "Unit1.MotionNodes".MotionToPLC.Status.StackMain.Busy.SemiStepBusy )
      I_Contact( "Unit1.MotionNodes".MotionToPLC.Status.StackMain.Busy.FullStepBusy )
      I_Contact( "Unit1.MotionNodes".MotionToPLC.Status.StackMain.Busy.AutoBusy )
      Not()
      Contact( "Unit1.Em4.ControlNodes".mainPnP.jobInterface.unloadJob3.workingDone )
      P_Trig( #statPulse.workingDone.mainPnP[51] )
      R_Coil( "Unit1.Em4.ControlNodes".mainPnP.jobInterface.unloadJob3.workingDone )
   END_RUNG
   RUNG wire#powerrail
      P_Contact(operand := #instMainPnPAvoidJob4.jobStatus.completed, bit := #statPulse.workingDone.mainPnP[0])
      S_Coil( "Unit1.Em4.ControlNodes".mainPnP.jobInterface.avoidJob4.workingDone )
   END_RUNG
   RUNG wire#powerrail
      P_Contact(operand := #instMainPnPOneLoadJob5.jobStatus.completed, bit := #statPulse.workingDone.mainPnP[1])
      S_Coil( "Unit1.Em4.ControlNodes".mainPnP.jobInterface.oneLoadJob5.workingDone )
   END_RUNG
   RUNG wire#powerrail
      P_Contact(operand := #instMainPnPOneUnLoadJob6.jobStatus.completed, bit := #statPulse.workingDone.mainPnP[2])
      wire#w5
      R_Coil( "Unit1.Em4.ControlNodes".mainPnP.jobInterface.avoidJob4.workingDone )
      R_Coil( "Unit1.Em4.ControlNodes".mainPnP.jobInterface.oneLoadJob5.workingDone )
   END_RUNG
   RUNG wire#powerrail
      I_Contact( #unitStatus.specialFunctions.dryRun )
      Contact( "Unit1.Em4.ControlNodes".cmAnodeMainPnP1SuctionPlateVacuum.monitoring.inHomePos )
      wire#w6
      P_Trig( #statPulse.workingDone.mainPnP[3] )
   END_RUNG wire#w5
   RUNG wire#powerrail
      Contact( #unitStatus.specialFunctions.dryRun )
      Contact( #statUnitStatus.state.idle )
   END_RUNG wire#w6
   RUNG wire#powerrail
      Contact( #instMainPnPOneUnLoadJob6.jobStatus.completed )
      Coil( "Unit1.Em4.ControlNodes".mainPnP.jobInterface.oneUnLoadJob6.workingDone )
   END_RUNG
   // the same network as SCL:
   "Unit1.Em4.ControlNodes".mainPnP.jobInterface.homeJob10.workingDone := #instMainPnPHomeJob10.jobStatus.completed;
   #_w1 := #instMainPnPLoadJob2.jobStatus.completed AND NOT #statPulse.workingDone.mainPnP[20];   // rising edge of #instMainPnPLoadJob2.jobStatus.completed
   #statPulse.workingDone.mainPnP[20] := #instMainPnPLoadJob2.jobStatus.completed;
   IF #_w1 THEN "Unit1.Em4.ControlNodes".mainPnP.jobInterface.loadJob2.workingDone := TRUE; END_IF;
   #_w2 := #instMainPnPUnloadJob3.jobStatus.completed AND NOT #statPulse.workingDone.mainPnP[30];   // rising edge of #instMainPnPUnloadJob3.jobStatus.completed
   #statPulse.workingDone.mainPnP[30] := #instMainPnPUnloadJob3.jobStatus.completed;
   #_w3 := ("Unit1.EmData".currentTotalElectrode = 0) AND #statUnitStatus.state.execute AND NOT "Unit1.MotionNodes".MotionToPLC.Status.StackMain.Busy.SemiStepBusy AND NOT "Unit1.MotionNodes".MotionToPLC.Status.StackMain.Busy.FullStepBusy AND NOT "Unit1.MotionNodes".MotionToPLC.Status.StackMain.Busy.AutoBusy AND "Unit1.Em4.ControlNodes".cmAnodeAlignTableSuctionPlateVacuum.monitoring.inWorkPos AND "Unit1.Em4.ControlNodes".cmAnodeMainPnP1SuctionPlateVacuum.monitoring.inHomePos AND "Unit1.Em4.ControlNodes".cmAnodeMainPnP2SuctionPlateVacuum.monitoring.inHomePos;
   #_w4 := #_w3 AND NOT #statPulse.workingDone.mainPnP[32];   // rising edge
   #statPulse.workingDone.mainPnP[32] := #_w3;
   #_w5 := (NOT (NOT "Unit1.Em4.ControlNodes".cmAnodeMainPnP1SuctionPlateVacuum.monitoring.inHomePos AND NOT "Unit1.Em4.ControlNodes".cmAnodeMainPnP2SuctionPlateVacuum.monitoring.inHomePos) AND NOT #unitStatus.specialFunctions.dryRun) OR (#unitStatus.specialFunctions.dryRun AND #statUnitStatus.state.idle);
   #_w6 := #_w5 AND NOT #statPulse.workingDone.mainPnP[31];   // rising edge
   #statPulse.workingDone.mainPnP[31] := #_w5;
   IF #_w2 OR #_w4 OR #_w6 THEN
       "Unit1.Em4.ControlNodes".mainPnP.jobInterface.loadJob2.workingDone := FALSE;
   END_IF;
   #_w7 := #instMainPnPUnloadJob3.jobStatus.completed AND ("Unit1.MotionNodes".MotionToPLC.Status.StackMain.Busy.SemiStepBusy OR "Unit1.MotionNodes".MotionToPLC.Status.StackMain.Busy.FullStepBusy OR "Unit1.MotionNodes".MotionToPLC.Status.StackMain.Busy.AutoBusy);
   #_w8 := #_w7 AND NOT #statPulse.workingDone.mainPnP[52];   // rising edge
   #statPulse.workingDone.mainPnP[52] := #_w7;
   IF #_w8 THEN "Unit1.Em4.ControlNodes".mainPnP.jobInterface.unloadJob3.workingDone := TRUE; END_IF;
   #_w9 := NOT (NOT "Unit1.MotionNodes".MotionToPLC.Status.StackMain.Busy.SemiStepBusy AND NOT "Unit1.MotionNodes".MotionToPLC.Status.StackMain.Busy.FullStepBusy AND NOT "Unit1.MotionNodes".MotionToPLC.Status.StackMain.Busy.AutoBusy) AND "Unit1.Em4.ControlNodes".mainPnP.jobInterface.unloadJob3.workingDone;
   #_w10 := #_w9 AND NOT #statPulse.workingDone.mainPnP[51];   // rising edge
   #statPulse.workingDone.mainPnP[51] := #_w9;
   IF #_w10 THEN "Unit1.Em4.ControlNodes".mainPnP.jobInterface.unloadJob3.workingDone := FALSE; END_IF;
   #_w11 := #instMainPnPAvoidJob4.jobStatus.completed AND NOT #statPulse.workingDone.mainPnP[0];   // rising edge of #instMainPnPAvoidJob4.jobStatus.completed
   #statPulse.workingDone.mainPnP[0] := #instMainPnPAvoidJob4.jobStatus.completed;
   IF #_w11 THEN "Unit1.Em4.ControlNodes".mainPnP.jobInterface.avoidJob4.workingDone := TRUE; END_IF;
   #_w12 := #instMainPnPOneLoadJob5.jobStatus.completed AND NOT #statPulse.workingDone.mainPnP[1];   // rising edge of #instMainPnPOneLoadJob5.jobStatus.completed
   #statPulse.workingDone.mainPnP[1] := #instMainPnPOneLoadJob5.jobStatus.completed;
   IF #_w12 THEN "Unit1.Em4.ControlNodes".mainPnP.jobInterface.oneLoadJob5.workingDone := TRUE; END_IF;
   #_w13 := #instMainPnPOneUnLoadJob6.jobStatus.completed AND NOT #statPulse.workingDone.mainPnP[2];   // rising edge of #instMainPnPOneUnLoadJob6.jobStatus.completed
   #statPulse.workingDone.mainPnP[2] := #instMainPnPOneUnLoadJob6.jobStatus.completed;
   #_w14 := (NOT #unitStatus.specialFunctions.dryRun AND "Unit1.Em4.ControlNodes".cmAnodeMainPnP1SuctionPlateVacuum.monitoring.inHomePos) OR (#unitStatus.specialFunctions.dryRun AND #statUnitStatus.state.idle);
   #_w15 := #_w14 AND NOT #statPulse.workingDone.mainPnP[3];   // rising edge
   #statPulse.workingDone.mainPnP[3] := #_w14;
   IF #_w13 OR #_w15 THEN
       "Unit1.Em4.ControlNodes".mainPnP.jobInterface.avoidJob4.workingDone := FALSE;
       "Unit1.Em4.ControlNodes".mainPnP.jobInterface.oneLoadJob5.workingDone := FALSE;
   END_IF;
   "Unit1.Em4.ControlNodes".mainPnP.jobInterface.oneUnLoadJob6.workingDone := #instMainPnPOneUnLoadJob6.jobStatus.completed;
END_REGION

